LIN {X 0,Y 497.029,Z 1160.432,A -85,B 0,C 180,E1 21832.452,E2 21832.452} C_VEL
LIN {X 0,Y 502.234,Z 1141.982,A -85,B 0,C 180,E1 21830.218,E2 21830.218} C_VEL
LIN {X 0,Y 508.212,Z 1120.317,A -85,B 0,C 180,E1 21827.949,E2 21827.949} C_VEL
LIN {X 0,Y 512.986,Z 1102.562,A -85,B 0,C 180,E1 21826.314,E2 21826.314} C_VEL
LIN {X 0,Y 517.599,Z 1084.829,A -85,B 0,C 180,E1 21824.86,E2 21824.86} C_VEL
LIN {X 0,Y 522.261,Z 1066.052,A -85,B 0,C 180,E1 21823.491,E2 21823.491} C_VEL
LIN {X 0,Y 527.633,Z 1043.21,A -85,B 0,C 180,E1 21822.036,E2 21822.036} C_VEL
LIN {X 0,Y 533.047,Z 1017.477,A -85,B 0,C 180,E1 21820.656,E2 21820.656} C_VEL
LIN {X 0,Y 537.035,Z 996.541,A -85,B 0,C 180,E1 21819.707,E2 21819.707} C_VEL
LIN {X 0,Y 540.556,Z 975.901,A -85,B 0,C 180,E1 21818.909,E2 21818.909} C_VEL
LIN {X 0,Y 543.808,Z 954.173,A -85,B 0,C 180,E1 21818.206,E2 21818.206} C_VEL
LIN {X 0,Y 547.16,Z 927.563,A -85,B 0,C 180,E1 21817.516,E2 21817.516} C_VEL
LIN {X 0,Y 549.546,Z 900.175,A -85,B 0,C 180,E1 21816.999,E2 21816.999} C_VEL
LIN {X 0,Y 555.879,Z 766.866,A -85,B 0,C 180,E1 21814.975,E2 21814.975} C_VEL
LIN {X 0,Y 566.177,Z 554.638,A -85,B 0,C 180,E1 21811.749,E2 21811.749} C_VEL
LIN {X 0,Y 566.782,Z 540.369,A -85,B 0,C 180,E1 21811.512,E2 21811.512} C_VEL
LIN {X 0,Y 555.133,Z 521.953,A -85,B 0,C 180,E1 21809.04,E2 21809.04} C_VEL
LIN {X 0,Y 545.079,Z 507.132,A -85,B 0,C 180,E1 21806.678,E2 21806.678} C_VEL
LIN {X 0,Y 535.268,Z 493.183,A -85,B 0,C 180,E1 21804.09,E2 21804.09} C_VEL
LIN {X 0,Y 527.729,Z 483.129,A -85,B 0,C 180,E1 21801.858,E2 21801.858} C_VEL
LIN {X 0,Y 523.599,Z 477.699,A -85,B 0,C 180,E1 21800.513,E2 21800.513} C_VEL
LIN {X 0,Y 518.429,Z 471.033,A -85,B 0,C 180,E1 21798.673,E2 21798.673} C_VEL
LIN {X 0,Y 515.934,Z 468.011,A -85,B 0,C 180,E1 21797.714,E2 21797.714} C_VEL
LIN {X 0,Y 512.62,Z 464.186,A -85,B 0,C 180,E1 21796.352,E2 21796.352} C_VEL
LIN {X 0,Y 511.594,Z 462.527,A -85,B 0,C 180,E1 21795.88,E2 21795.88} C_VEL
LIN {X 0,Y 508.237,Z 459.547,A -85,B 0,C 180,E1 21794.353,E2 21794.353} C_VEL
LIN {X 0,Y 505.989,Z 456.089,A -85,B 0,C 180,E1 21793.135,E2 21793.135} C_VEL
LIN {X 0,Y 502.714,Z 453.695,A -85,B 0,C 180,E1 21791.298,E2 21791.298} C_VEL
LIN {X 0,Y 500.503,Z 449.64,A -85,B 0,C 180,E1 21789.661,E2 21789.661} C_VEL
LIN {X 0,Y 496.627,Z 447.233,A -85,B 0,C 180,E1 21786.358,E2 21786.358} C_VEL
LIN {X 0,Y 494.773,Z 443.193,A -85,B 0,C 180,E1 21783.302,E2 21783.302} C_VEL
LIN {X 0,Y 493.904,Z 442.834,A -85,B 0,C 180,E1 21780.464,E2 21780.464} C_VEL
LIN {X 0,Y 494.784,Z 443.176,A -85,B 0,C 180,E1 21776.176,E2 21776.176} C_VEL
LIN {X 0,Y 496.308,Z 446.772,A -85,B 0,C 180,E1 21773.522,E2 21773.522} C_VEL
LIN {X 0,Y 499.957,Z 449.46,A -85,B 0,C 180,E1 21770.212,E2 21770.212} C_VEL
LIN {X 0,Y 500.671,Z 449.883,A -85,B 0,C 180,E1 21769.704,E2 21769.704} C_VEL
LIN {X 0,Y 502.481,Z 453.39,A -85,B 0,C 180,E1 21768.347,E2 21768.347} C_VEL
LIN {X 0,Y 506.131,Z 456.157,A -85,B 0,C 180,E1 21766.286,E2 21766.286} C_VEL
LIN {X 0,Y 509.284,Z 460.773,A -85,B 0,C 180,E1 21764.63,E2 21764.63} C_VEL
LIN {X 0,Y 511.991,Z 463.084,A -85,B 0,C 180,E1 21763.433,E2 21763.433} C_VEL
LIN {X 0,Y 515.015,Z 467.149,A -85,B 0,C 180,E1 21762.136,E2 21762.136} C_VEL
LIN {X 0,Y 517.324,Z 469.281,A -85,B 0,C 180,E1 21761.256,E2 21761.256} C_VEL
LIN {X 0,Y 520.829,Z 473.673,A -85,B 0,C 180,E1 21759.959,E2 21759.959} C_VEL
LIN {X 0,Y 522.505,Z 475.511,A -85,B 0,C 180,E1 21759.383,E2 21759.383} C_VEL
LIN {X 0,Y 526.451,Z 480.194,A -85,B 0,C 180,E1 21758.086,E2 21758.086} C_VEL
LIN {X 0,Y 532.504,Z 487.779,A -85,B 0,C 180,E1 21756.248,E2 21756.248} C_VEL
LIN {X 0,Y 537.349,Z 493.885,A -85,B 0,C 180,E1 21754.896,E2 21754.896} C_VEL
LIN {X 0,Y 544.214,Z 502.496,A -85,B 0,C 180,E1 21753.129,E2 21753.129} C_VEL
LIN {X 0,Y 555.457,Z 517.635,A -85,B 0,C 180,E1 21750.506,E2 21750.506} C_VEL
LIN {X 0,Y 566.795,Z 533.76,A -85,B 0,C 180,E1 21748.135,E2 21748.135} C_VEL
LIN {X 0,Y 556.148,Z 750.221,A -85,B 0,C 180,E1 21744.845,E2 21744.845} C_VEL
LIN {X 0,Y 549.972,Z 878.471,A -85,B 0,C 180,E1 21742.897,E2 21742.897} C_VEL
LIN {X 0,Y 547.763,Z 904.531,A -85,B 0,C 180,E1 21742.395,E2 21742.395} C_VEL
LIN {X 0,Y 544.492,Z 931.574,A -85,B 0,C 180,E1 21741.681,E2 21741.681} C_VEL
LIN {X 0,Y 541.398,Z 952.771,A -85,B 0,C 180,E1 21740.982,E2 21740.982} C_VEL
LIN {X 0,Y 538.057,Z 972.694,A -85,B 0,C 180,E1 21740.201,E2 21740.201} C_VEL
LIN {X 0,Y 534.237,Z 992.896,A -85,B 0,C 180,E1 21739.277,E2 21739.277} C_VEL
LIN {X 0,Y 529.413,Z 1016.049,A -85,B 0,C 180,E1 21738.041,E2 21738.041} C_VEL
LIN {X 0,Y 523.704,Z 1040.347,A -85,B 0,C 180,E1 21736.501,E2 21736.501} C_VEL
LIN {X 0,Y 518.815,Z 1059.671,A -85,B 0,C 180,E1 21735.083,E2 21735.083} C_VEL
LIN {X 0,Y 514.02,Z 1077.682,A -85,B 0,C 180,E1 21733.587,E2 21733.587} C_VEL
LIN {X 0,Y 509.135,Z 1095.319,A -85,B 0,C 180,E1 21731.935,E2 21731.935} C_VEL
LIN {X 0,Y 503.229,Z 1115.953,A -85,B 0,C 180,E1 21729.74,E2 21729.74} C_VEL
LIN {X 0,Y 498.603,Z 1131.683,A -85,B 0,C 180,E1 21727.817,E2 21727.817} C_VEL
LIN {X 0,Y 496.227,Z 1136.911,A -85,B 0,C 180,E1 21727.204,E2 21727.204} C_VEL
LIN {X 0,Y 486.897,Z 1150.907,A -85,B 0,C 180,E1 21725.694,E2 21725.694} C_VEL
LIN {X 0,Y 485.066,Z 1155.035,A -85,B 0,C 180,E1 21725.127,E2 21725.127} C_VEL
LIN {X 0,Y 480.071,Z 1171.483,A -85,B 0,C 180,E1 21722.354,E2 21722.354} C_VEL
LIN {X 0,Y 476.443,Z 1184.012,A -85,B 0,C 180,E1 21719.957,E2 21719.957} C_VEL
LIN {X 0,Y 473.338,Z 1195.518,A -85,B 0,C 180,E1 21717.474,E2 21717.474} C_VEL
LIN {X 0,Y 470.207,Z 1208.206,A -85,B 0,C 180,E1 21714.357,E2 21714.357} C_VEL
LIN {X 0,Y 467.788,Z 1219.059,A -85,B 0,C 180,E1 21711.169,E2 21711.169} C_VEL
LIN {X 0,Y 466.306,Z 1226.894,A -85,B 0,C 180,E1 21708.496,E2 21708.496} C_VEL
LIN {X 0,Y 465.289,Z 1233.576,A -85,B 0,C 180,E1 21705.831,E2 21705.831} C_VEL
LIN {X 0,Y 464.545,Z 1239.653,A -85,B 0,C 180,E1 21702.929,E2 21702.929} C_VEL
LIN {X 0,Y 464.073,Z 1245.171,A -85,B 0,C 180,E1 21699.543,E2 21699.543} C_VEL
LIN {X 0,Y 463.961,Z 1248.712,A -85,B 0,C 180,E1 21696.529,E2 21696.529} C_VEL
LIN {X 0,Y 463.915,Z 1250.719,A -85,B 0,C 180,E1 21693.949,E2 21693.949} C_VEL
LIN {X 0,Y 463.904,Z 1251.727,A -85,B 0,C 180,E1 21691.476,E2 21691.476} C_VEL
LIN {X 0,Y 463.872,Z 1251.832,A -85,B 0,C 180,E1 21689.006,E2 21689.006} C_VEL
LIN {X 0,Y 463.913,Z 1251.035,A -85,B 0,C 180,E1 21686.535,E2 21686.535} C_VEL
LIN {X 0,Y 463.95,Z 1249.219,A -85,B 0,C 180,E1 21683.933,E2 21683.933} C_VEL
LIN {X 0,Y 464.051,Z 1246.391,A -85,B 0,C 180,E1 21681.32,E2 21681.32} C_VEL
LIN {X 0,Y 464.326,Z 1242,A -85,B 0,C 180,E1 21678.316,E2 21678.316} C_VEL
LIN {X 0,Y 465.026,Z 1235.477,A -85,B 0,C 180,E1 21674.892,E2 21674.892} C_VEL
LIN {X 0,Y 466.1,Z 1228.126,A -85,B 0,C 180,E1 21671.868,E2 21671.868} C_VEL
LIN {X 0,Y 467.52,Z 1220.38,A -85,B 0,C 180,E1 21669.167,E2 21669.167} C_VEL
LIN {X 0,Y 469.256,Z 1212.057,A -85,B 0,C 180,E1 21666.647,E2 21666.647} C_VEL
LIN {X 0,Y 471.63,Z 1202.142,A -85,B 0,C 180,E1 21664.016,E2 21664.016} C_VEL
LIN {X 0,Y 475.367,Z 1188.092,A -85,B 0,C 180,E1 21660.787,E2 21660.787} C_VEL
LIN {X 0,Y 479.151,Z 1174.611,A -85,B 0,C 180,E1 21658.128,E2 21658.128} C_VEL
LIN {X 0,Y 482.964,Z 1161.693,A -85,B 0,C 180,E1 21655.867,E2 21655.867} C_VEL
LIN {X 0,Y 487.08,Z 1148.162,A -85,B 0,C 180,E1 21653.753,E2 21653.753} C_VEL
LIN {X 0,Y 492.267,Z 1131.357,A -85,B 0,C 180,E1 21651.418,E2 21651.418} C_VEL
LIN {X 0,Y 498.504,Z 1110.82,A -85,B 0,C 180,E1 21648.954,E2 21648.954} C_VEL
LIN {X 0,Y 503.601,Z 1093.635,A -85,B 0,C 180,E1 21647.15,E2 21647.15} C_VEL
LIN {X 0,Y 508.295,Z 1077.31,A -85,B 0,C 180,E1 21645.624,E2 21645.624} C_VEL
LIN {X 0,Y 513.079,Z 1059.953,A -85,B 0,C 180,E1 21644.176,E2 21644.176} C_VEL
LIN {X 0,Y 518.353,Z 1039.81,A -85,B 0,C 180,E1 21642.694,E2 21642.694} C_VEL
LIN {X 0,Y 524.566,Z 1013.892,A -85,B 0,C 180,E1 21641.069,E2 21641.069} C_VEL
LIN {X 0,Y 529.021,Z 993.124,A -85,B 0,C 180,E1 21639.962,E2 21639.962} C_VEL
LIN {X 0,Y 532.958,Z 972.91,A -85,B 0,C 180,E1 21639.036,E2 21639.036} C_VEL
LIN {X 0,Y 536.564,Z 952.039,A -85,B 0,C 180,E1 21638.22,E2 21638.22} C_VEL
LIN {X 0,Y 540.132,Z 928.072,A -85,B 0,C 180,E1 21637.442,E2 21637.442} C_VEL
LIN {X 0,Y 543.36,Z 900.216,A -85,B 0,C 180,E1 21636.745,E2 21636.745} C_VEL
LIN {X 0,Y 545.306,Z 877.407,A -85,B 0,C 180,E1 21636.317,E2 21636.317} C_VEL
LIN {X 0,Y 555.554,Z 671.599,A -85,B 0,C 180,E1 21633.181,E2 21633.181} C_VEL
LIN {X 0,Y 562.367,Z 538.21,A -85,B 0,C 180,E1 21631.128,E2 21631.128} C_VEL
LIN {X 0,Y 551.699,Z 522.97,A -85,B 0,C 180,E1 21628.822,E2 21628.822} C_VEL
LIN {X 0,Y 541.383,Z 508.945,A -85,B 0,C 180,E1 21626.342,E2 21626.342} C_VEL
LIN {X 0,Y 532.518,Z 497.635,A -85,B 0,C 180,E1 21623.957,E2 21623.957} C_VEL
LIN {X 0,Y 528.303,Z 492.352,A -85,B 0,C 180,E1 21622.712,E2 21622.712} C_VEL
LIN {X 0,Y 524.222,Z 487.316,A -85,B 0,C 180,E1 21621.424,E2 21621.424} C_VEL
LIN {X 0,Y 519.631,Z 481.696,A -85,B 0,C 180,E1 21619.854,E2 21619.854} C_VEL
LIN {X 0,Y 515.928,Z 477.216,A -85,B 0,C 180,E1 21618.474,E2 21618.474} C_VEL
LIN {X 0,Y 514.556,Z 475.732,A -85,B 0,C 180,E1 21617.939,E2 21617.939} C_VEL
LIN {X 0,Y 511.083,Z 471.685,A -85,B 0,C 180,E1 21616.48,E2 21616.48} C_VEL
LIN {X 0,Y 509.897,Z 470.059,A -85,B 0,C 180,E1 21615.934,E2 21615.934} C_VEL
LIN {X 0,Y 506.547,Z 466.804,A -85,B 0,C 180,E1 21614.343,E2 21614.343} C_VEL
LIN {X 0,Y 504.877,Z 463.969,A -85,B 0,C 180,E1 21613.398,E2 21613.398} C_VEL
LIN {X 0,Y 501.485,Z 461.38,A -85,B 0,C 180,E1 21611.443,E2 21611.443} C_VEL
LIN {X 0,Y 499.477,Z 457.698,A -85,B 0,C 180,E1 21609.914,E2 21609.914} C_VEL
LIN {X 0,Y 495.09,Z 454.362,A -85,B 0,C 180,E1 21605.796,E2 21605.796} C_VEL
LIN {X 0,Y 493.761,Z 450.858,A -85,B 0,C 180,E1 21603.018,E2 21603.018} C_VEL
LIN {X 0,Y 493.831,Z 450.948,A -85,B 0,C 180,E1 21597.215,E2 21597.215} C_VEL
LIN {X 0,Y 495.777,Z 455.253,A -85,B 0,C 180,E1 21593.748,E2 21593.748} C_VEL
LIN {X 0,Y 499.49,Z 457.7,A -85,B 0,C 180,E1 21590.494,E2 21590.494} C_VEL
LIN {X 0,Y 501.581,Z 461.525,A -85,B 0,C 180,E1 21588.909,E2 21588.909} C_VEL
LIN {X 0,Y 505.181,Z 464.453,A -85,B 0,C 180,E1 21586.843,E2 21586.843} C_VEL
LIN {X 0,Y 507.875,Z 468.4,A -85,B 0,C 180,E1 21585.404,E2 21585.404} C_VEL
LIN {X 0,Y 510.518,Z 470.754,A -85,B 0,C 180,E1 21584.202,E2 21584.202} C_VEL
LIN {X 0,Y 513.616,Z 474.922,A -85,B 0,C 180,E1 21582.846,E2 21582.846} C_VEL
LIN {X 0,Y 515.651,Z 477.08,A -85,B 0,C 180,E1 21582.042,E2 21582.042} C_VEL
LIN {X 0,Y 519.586,Z 482.261,A -85,B 0,C 180,E1 21580.554,E2 21580.554} C_VEL
LIN {X 0,Y 523.665,Z 487.63,A -85,B 0,C 180,E1 21579.139,E2 21579.139} C_VEL
LIN {X 0,Y 528.756,Z 494.46,A -85,B 0,C 180,E1 21577.514,E2 21577.514} C_VEL
LIN {X 0,Y 534.895,Z 503.025,A -85,B 0,C 180,E1 21575.716,E2 21575.716} C_VEL
LIN {X 0,Y 543.878,Z 515.818,A -85,B 0,C 180,E1 21573.347,E2 21573.347} C_VEL
LIN {X 0,Y 554.813,Z 532.468,A -85,B 0,C 180,E1 21570.764,E2 21570.764} C_VEL
LIN {X 0,Y 562.515,Z 545.109,A -85,B 0,C 180,E1 21569.096,E2 21569.096} C_VEL
LIN {X 0,Y 551.791,Z 757.323,A -85,B 0,C 180,E1 21565.855,E2 21565.855} C_VEL
LIN {X 0,Y 544.786,Z 899.692,A -85,B 0,C 180,E1 21563.684,E2 21563.684} C_VEL
LIN {X 0,Y 542.427,Z 926.225,A -85,B 0,C 180,E1 21563.184,E2 21563.184} C_VEL
LIN {X 0,Y 538.96,Z 953.287,A -85,B 0,C 180,E1 21562.491,E2 21562.491} C_VEL
LIN {X 0,Y 535.662,Z 974.729,A -85,B 0,C 180,E1 21561.803,E2 21561.803} C_VEL
LIN {X 0,Y 532.026,Z 995.532,A -85,B 0,C 180,E1 21561.002,E2 21561.002} C_VEL
LIN {X 0,Y 527.885,Z 1016.607,A -85,B 0,C 180,E1 21560.05,E2 21560.05} C_VEL
LIN {X 0,Y 522.429,Z 1041.913,A -85,B 0,C 180,E1 21558.699,E2 21558.699} C_VEL
LIN {X 0,Y 516.806,Z 1065.056,A -85,B 0,C 180,E1 21557.227,E2 21557.227} C_VEL
LIN {X 0,Y 512.008,Z 1083.719,A -85,B 0,C 180,E1 21555.867,E2 21555.867} C_VEL
LIN {X 0,Y 507.226,Z 1101.42,A -85,B 0,C 180,E1 21554.415,E2 21554.415} C_VEL
LIN {X 0,Y 502.213,Z 1119.333,A -85,B 0,C 180,E1 21552.763,E2 21552.763} C_VEL
LIN {X 0,Y 496.243,Z 1140.304,A -85,B 0,C 180,E1 21550.569,E2 21550.569} C_VEL
LIN {X 0,Y 490.533,Z 1159.602,A -85,B 0,C 180,E1 21548.221,E2 21548.221} C_VEL
LIN {X 0,Y 486.187,Z 1174.525,A -85,B 0,C 180,E1 21546.178,E2 21546.178} C_VEL
LIN {X 0,Y 482.185,Z 1188.461,A -85,B 0,C 180,E1 21544.052,E2 21544.052} C_VEL
LIN {X 0,Y 478.313,Z 1202.513,A -85,B 0,C 180,E1 21541.653,E2 21541.653} C_VEL
LIN {X 0,Y 473.954,Z 1219.168,A -85,B 0,C 180,E1 21538.389,E2 21538.389} C_VEL
LIN {X 0,Y 471.191,Z 1230.65,A -85,B 0,C 180,E1 21535.791,E2 21535.791} C_VEL
LIN {X 0,Y 468.998,Z 1240.65,A -85,B 0,C 180,E1 21533.234,E2 21533.234} C_VEL
LIN {X 0,Y 467.323,Z 1249.445,A -85,B 0,C 180,E1 21530.678,E2 21530.678} C_VEL
LIN {X 0,Y 465.884,Z 1258.181,A -85,B 0,C 180,E1 21527.749,E2 21527.749} C_VEL
LIN {X 0,Y 464.794,Z 1266.563,A -85,B 0,C 180,E1 21524.328,E2 21524.328} C_VEL
LIN {X 0,Y 464.305,Z 1272.056,A -85,B 0,C 180,E1 21521.52,E2 21521.52} C_VEL
LIN {X 0,Y 464.051,Z 1276.014,A -85,B 0,C 180,E1 21518.93,E2 21518.93} C_VEL
LIN {X 0,Y 463.958,Z 1278.95,A -85,B 0,C 180,E1 21516.316,E2 21516.316} C_VEL
LIN {X 0,Y 463.916,Z 1280.806,A -85,B 0,C 180,E1 21513.836,E2 21513.836} C_VEL
LIN {X 0,Y 463.896,Z 1281.756,A -85,B 0,C 180,E1 21511.364,E2 21511.364} C_VEL
LIN {X 0,Y 463.881,Z 1281.803,A -85,B 0,C 180,E1 21508.894,E2 21508.894} C_VEL
LIN {X 0,Y 463.913,Z 1280.948,A -85,B 0,C 180,E1 21506.422,E2 21506.422} C_VEL
LIN {X 0,Y 463.949,Z 1279.187,A -85,B 0,C 180,E1 21503.944,E2 21503.944} C_VEL
LIN {X 0,Y 464.051,Z 1276.347,A -85,B 0,C 180,E1 21501.331,E2 21501.331} C_VEL
LIN {X 0,Y 464.262,Z 1272.648,A -85,B 0,C 180,E1 21498.83,E2 21498.83} C_VEL
LIN {X 0,Y 464.68,Z 1267.896,A -85,B 0,C 180,E1 21496.315,E2 21496.315} C_VEL
LIN {X 0,Y 465.38,Z 1261.818,A -85,B 0,C 180,E1 21493.66,E2 21493.66} C_VEL
LIN {X 0,Y 466.562,Z 1253.866,A -85,B 0,C 180,E1 21490.736,E2 21490.736} C_VEL
LIN {X 0,Y 468.621,Z 1242.575,A -85,B 0,C 180,E1 21487.289,E2 21487.289} C_VEL
LIN {X 0,Y 470.829,Z 1232.284,A -85,B 0,C 180,E1 21484.605,E2 21484.605} C_VEL
LIN {X 0,Y 473.308,Z 1221.766,A -85,B 0,C 180,E1 21482.176,E2 21482.176} C_VEL
LIN {X 0,Y 476.286,Z 1209.997,A -85,B 0,C 180,E1 21479.754,E2 21479.754} C_VEL
LIN {X 0,Y 480.497,Z 1194.732,A -85,B 0,C 180,E1 21476.97,E2 21476.97} C_VEL
LIN {X 0,Y 485.421,Z 1177.178,A -85,B 0,C 180,E1 21474.206,E2 21474.206} C_VEL
LIN {X 0,Y 489.946,Z 1161.563,A -85,B 0,C 180,E1 21472.035,E2 21472.035} C_VEL
LIN {X 0,Y 494.553,Z 1145.778,A -85,B 0,C 180,E1 21470.074,E2 21470.074} C_VEL
LIN {X 0,Y 500.556,Z 1125.32,A -85,B 0,C 180,E1 21467.825,E2 21467.825} C_VEL
LIN {X 0,Y 506.453,Z 1104.21,A -85,B 0,C 180,E1 21465.829,E2 21465.829} C_VEL
LIN {X 0,Y 511.371,Z 1086.037,A -85,B 0,C 180,E1 21464.315,E2 21464.315} C_VEL
LIN {X 0,Y 516.177,Z 1067.413,A -85,B 0,C 180,E1 21462.938,E2 21462.938} C_VEL
LIN {X 0,Y 521.032,Z 1047.472,A -85,B 0,C 180,E1 21461.64,E2 21461.64} C_VEL
LIN {X 0,Y 526.618,Z 1022.881,A -85,B 0,C 180,E1 21460.258,E2 21460.258} C_VEL
LIN {X 0,Y 531.493,Z 998.254,A -85,B 0,C 180,E1 21459.114,E2 21459.114} C_VEL
LIN {X 0,Y 535.242,Z 977.114,A -85,B 0,C 180,E1 21458.285,E2 21458.285} C_VEL
LIN {X 0,Y 538.532,Z 955.967,A -85,B 0,C 180,E1 21457.591,E2 21457.591} C_VEL
LIN {X 0,Y 541.423,Z 934.088,A -85,B 0,C 180,E1 21457.003,E2 21457.003} C_VEL
LIN {X 0,Y 544.311,Z 906.44,A -85,B 0,C 180,E1 21456.43,E2 21456.43} C_VEL
LIN {X 0,Y 546.777,Z 860.87,A -85,B 0,C 180,E1 21455.715,E2 21455.715} C_VEL
LIN {X 0,Y 557.422,Z 642.939,A -85,B 0,C 180,E1 21452.406,E2 21452.406} C_VEL
LIN {X 0,Y 562.394,Z 544.765,A -85,B 0,C 180,E1 21450.889,E2 21450.889} C_VEL
LIN {X 0,Y 551.819,Z 527.929,A -85,B 0,C 180,E1 21448.579,E2 21448.579} C_VEL
LIN {X 0,Y 542.426,Z 513.869,A -85,B 0,C 180,E1 21446.317,E2 21446.317} C_VEL
LIN {X 0,Y 532.943,Z 500.218,A -85,B 0,C 180,E1 21443.76,E2 21443.76} C_VEL
LIN {X 0,Y 525.603,Z 490.294,A -85,B 0,C 180,E1 21441.54,E2 21441.54} C_VEL
LIN {X 0,Y 521.54,Z 484.891,A -85,B 0,C 180,E1 21440.188,E2 21440.188} C_VEL
LIN {X 0,Y 516.605,Z 478.402,A -85,B 0,C 180,E1 21438.39,E2 21438.39} C_VEL
LIN {X 0,Y 514.143,Z 475.469,A -85,B 0,C 180,E1 21437.427,E2 21437.427} C_VEL
LIN {X 0,Y 510.824,Z 471.415,A -85,B 0,C 180,E1 21436.021,E2 21436.021} C_VEL
LIN {X 0,Y 509.874,Z 470.095,A -85,B 0,C 180,E1 21435.585,E2 21435.585} C_VEL
LIN {X 0,Y 506.394,Z 466.67,A -85,B 0,C 180,E1 21433.939,E2 21433.939} C_VEL
LIN {X 0,Y 504.598,Z 463.872,A -85,B 0,C 180,E1 21432.939,E2 21432.939} C_VEL
LIN {X 0,Y 501.39,Z 461.389,A -85,B 0,C 180,E1 21431.095,E2 21431.095} C_VEL
LIN {X 0,Y 499.213,Z 457.481,A -85,B 0,C 180,E1 21429.453,E2 21429.453} C_VEL
LIN {X 0,Y 495.356,Z 454.892,A -85,B 0,C 180,E1 21426.025,E2 21426.025} C_VEL
LIN {X 0,Y 493.629,Z 450.851,A -85,B 0,C 180,E1 21422.903,E2 21422.903} C_VEL
LIN {X 0,Y 493.719,Z 450.879,A -85,B 0,C 180,E1 21416.4,E2 21416.4} C_VEL
LIN {X 0,Y 495.239,Z 454.651,A -85,B 0,C 180,E1 21413.624,E2 21413.624} C_VEL
LIN {X 0,Y 498.995,Z 457.415,A -85,B 0,C 180,E1 21410.193,E2 21410.193} C_VEL
LIN {X 0,Y 499.518,Z 457.987,A -85,B 0,C 180,E1 21409.796,E2 21409.796} C_VEL
LIN {X 0,Y 501.418,Z 461.402,A -85,B 0,C 180,E1 21408.381,E2 21408.381} C_VEL
LIN {X 0,Y 505.141,Z 464.462,A -85,B 0,C 180,E1 21406.259,E2 21406.259} C_VEL
LIN {X 0,Y 507.741,Z 468.347,A -85,B 0,C 180,E1 21404.875,E2 21404.875} C_VEL
LIN {X 0,Y 510.458,Z 470.765,A -85,B 0,C 180,E1 21403.645,E2 21403.645} C_VEL
LIN {X 0,Y 513.648,Z 474.968,A -85,B 0,C 180,E1 21402.263,E2 21402.263} C_VEL
LIN {X 0,Y 515.651,Z 476.867,A -85,B 0,C 180,E1 21401.487,E2 21401.487} C_VEL
LIN {X 0,Y 519.419,Z 481.504,A -85,B 0,C 180,E1 21400.079,E2 21400.079} C_VEL
LIN {X 0,Y 521.209,Z 483.769,A -85,B 0,C 180,E1 21399.447,E2 21399.447} C_VEL
LIN {X 0,Y 525.787,Z 489.279,A -85,B 0,C 180,E1 21397.939,E2 21397.939} C_VEL
LIN {X 0,Y 530.484,Z 495.159,A -85,B 0,C 180,E1 21396.506,E2 21396.506} C_VEL
LIN {X 0,Y 535.454,Z 501.51,A -85,B 0,C 180,E1 21395.096,E2 21395.096} C_VEL
LIN {X 0,Y 541.963,Z 509.803,A -85,B 0,C 180,E1 21393.393,E2 21393.393} C_VEL
LIN {X 0,Y 552.775,Z 524.522,A -85,B 0,C 180,E1 21390.824,E2 21390.824} C_VEL
LIN {X 0,Y 562.381,Z 538.342,A -85,B 0,C 180,E1 21388.762,E2 21388.762} C_VEL
LIN {X 0,Y 551.332,Z 755.458,A -85,B 0,C 180,E1 21385.45,E2 21385.45} C_VEL
LIN {X 0,Y 545.179,Z 878.788,A -85,B 0,C 180,E1 21383.567,E2 21383.567} C_VEL
LIN {X 0,Y 542.874,Z 905.198,A -85,B 0,C 180,E1 21383.056,E2 21383.056} C_VEL
LIN {X 0,Y 539.515,Z 932.066,A -85,B 0,C 180,E1 21382.344,E2 21382.344} C_VEL
LIN {X 0,Y 536.337,Z 953.216,A -85,B 0,C 180,E1 21381.644,E2 21381.644} C_VEL
LIN {X 0,Y 532.92,Z 972.969,A -85,B 0,C 180,E1 21380.868,E2 21380.868} C_VEL
LIN {X 0,Y 528.987,Z 993.17,A -85,B 0,C 180,E1 21379.942,E2 21379.942} C_VEL
LIN {X 0,Y 524.098,Z 1015.92,A -85,B 0,C 180,E1 21378.725,E2 21378.725} C_VEL
LIN {X 0,Y 518.113,Z 1040.621,A -85,B 0,C 180,E1 21377.157,E2 21377.157} C_VEL
LIN {X 0,Y 513.081,Z 1059.873,A -85,B 0,C 180,E1 21375.737,E2 21375.737} C_VEL
LIN {X 0,Y 508.2,Z 1077.578,A -85,B 0,C 180,E1 21374.26,E2 21374.26} C_VEL
LIN {X 0,Y 503.244,Z 1094.82,A -85,B 0,C 180,E1 21372.641,E2 21372.641} C_VEL
LIN {X 0,Y 497.273,Z 1115.029,A -85,B 0,C 180,E1 21370.492,E2 21370.492} C_VEL
LIN {X 0,Y 491.355,Z 1134.185,A -85,B 0,C 180,E1 21368.114,E2 21368.114} C_VEL
LIN {X 0,Y 486.957,Z 1148.549,A -85,B 0,C 180,E1 21366.099,E2 21366.099} C_VEL
LIN {X 0,Y 485.066,Z 1155.035,A -85,B 0,C 180,E1 21365.127,E2 21365.127} C_VEL
LIN {X 0,Y 482.811,Z 1159.814,A -85,B 0,C 180,E1 21364.453,E2 21364.453} C_VEL
LIN {X 0,Y 473.489,Z 1172.374,A -85,B 0,C 180,E1 21362.728,E2 21362.728} C_VEL
LIN {X 0,Y 471.727,Z 1176.083,A -85,B 0,C 180,E1 21362.093,E2 21362.093} C_VEL
LIN {X 0,Y 466.996,Z 1192.12,A -85,B 0,C 180,E1 21358.791,E2 21358.791} C_VEL
LIN {X 0,Y 463.883,Z 1203.454,A -85,B 0,C 180,E1 21356.078,E2 21356.078} C_VEL
LIN {X 0,Y 461.498,Z 1212.969,A -85,B 0,C 180,E1 21353.487,E2 21353.487} C_VEL
LIN {X 0,Y 459.581,Z 1221.703,A -85,B 0,C 180,E1 21350.764,E2 21350.764} C_VEL
LIN {X 0,Y 457.834,Z 1231.194,A -85,B 0,C 180,E1 21347.272,E2 21347.272} C_VEL
LIN {X 0,Y 456.817,Z 1238.006,A -85,B 0,C 180,E1 21344.152,E2 21344.152} C_VEL
LIN {X 0,Y 456.332,Z 1242.744,A -85,B 0,C 180,E1 21341.495,E2 21341.495} C_VEL
LIN {X 0,Y 456.063,Z 1246.512,A -85,B 0,C 180,E1 21338.822,E2 21338.822} C_VEL
LIN {X 0,Y 455.957,Z 1249.28,A -85,B 0,C 180,E1 21336.162,E2 21336.162} C_VEL
LIN {X 0,Y 455.914,Z 1251.069,A -85,B 0,C 180,E1 21333.515,E2 21333.515} C_VEL
LIN {X 0,Y 455.872,Z 1251.893,A -85,B 0,C 180,E1 21330.874,E2 21330.874} C_VEL
LIN {X 0,Y 455.91,Z 1251.73,A -85,B 0,C 180,E1 21328.109,E2 21328.109} C_VEL
LIN {X 0,Y 455.928,Z 1250.234,A -85,B 0,C 180,E1 21324.836,E2 21324.836} C_VEL
LIN {X 0,Y 456.037,Z 1247.074,A -85,B 0,C 180,E1 21321.547,E2 21321.547} C_VEL
LIN {X 0,Y 456.285,Z 1243.268,A -85,B 0,C 180,E1 21318.748,E2 21318.748} C_VEL
LIN {X 0,Y 456.739,Z 1238.835,A -85,B 0,C 180,E1 21316.19,E2 21316.19} C_VEL
LIN {X 0,Y 457.498,Z 1233.141,A -85,B 0,C 180,E1 21313.489,E2 21313.489} C_VEL
LIN {X 0,Y 458.69,Z 1226.182,A -85,B 0,C 180,E1 21310.716,E2 21310.716} C_VEL
LIN {X 0,Y 460.854,Z 1215.914,A -85,B 0,C 180,E1 21307.277,E2 21307.277} C_VEL
LIN {X 0,Y 463.428,Z 1205.242,A -85,B 0,C 180,E1 21304.294,E2 21304.294} C_VEL
LIN {X 0,Y 466.258,Z 1194.672,A -85,B 0,C 180,E1 21301.705,E2 21301.705} C_VEL
LIN {X 0,Y 469.504,Z 1183.381,A -85,B 0,C 180,E1 21299.257,E2 21299.257} C_VEL
LIN {X 0,Y 473.822,Z 1169.379,A -85,B 0,C 180,E1 21296.575,E2 21296.575} C_VEL
LIN {X 0,Y 479.329,Z 1151.758,A -85,B 0,C 180,E1 21293.666,E2 21293.666} C_VEL
LIN {X 0,Y 484.037,Z 1136.973,A -85,B 0,C 180,E1 21291.528,E2 21291.528} C_VEL
LIN {X 0,Y 488.992,Z 1121.398,A -85,B 0,C 180,E1 21289.523,E2 21289.523} C_VEL
LIN {X 0,Y 494.706,Z 1103.27,A -85,B 0,C 180,E1 21287.458,E2 21287.458} C_VEL
LIN {X 0,Y 501.481,Z 1080.877,A -85,B 0,C 180,E1 21285.26,E2 21285.26} C_VEL
LIN {X 0,Y 506.836,Z 1062.205,A -85,B 0,C 180,E1 21283.669,E2 21283.669} C_VEL
LIN {X 0,Y 511.758,Z 1044.093,A -85,B 0,C 180,E1 21282.305,E2 21282.305} C_VEL
LIN {X 0,Y 516.855,Z 1024.083,A -85,B 0,C 180,E1 21280.982,E2 21280.982} C_VEL
LIN {X 0,Y 522.699,Z 998.992,A -85,B 0,C 180,E1 21279.56,E2 21279.56} C_VEL
LIN {X 0,Y 527.427,Z 975.719,A -85,B 0,C 180,E1 21278.464,E2 21278.464} C_VEL
LIN {X 0,Y 531.208,Z 954.707,A -85,B 0,C 180,E1 21277.626,E2 21277.626} C_VEL
LIN {X 0,Y 534.427,Z 934.083,A -85,B 0,C 180,E1 21276.934,E2 21276.934} C_VEL
LIN {X 0,Y 537.436,Z 911.189,A -85,B 0,C 180,E1 21276.307,E2 21276.307} C_VEL
LIN {X 0,Y 540.316,Z 881.853,A -85,B 0,C 180,E1 21275.702,E2 21275.702} C_VEL
LIN {X 0,Y 543.364,Z 825.579,A -85,B 0,C 180,E1 21274.827,E2 21274.827} C_VEL
LIN {X 0,Y 554.655,Z 606.621,A -85,B 0,C 180,E1 21271.485,E2 21271.485} C_VEL
LIN {X 0,Y 558.058,Z 542.861,A -85,B 0,C 180,E1 21270.498,E2 21270.498} C_VEL
LIN {X 0,Y 548.432,Z 529.017,A -85,B 0,C 180,E1 21268.355,E2 21268.355} C_VEL
LIN {X 0,Y 538.87,Z 515.862,A -85,B 0,C 180,E1 21266,E2 21266} C_VEL
LIN {X 0,Y 530.138,Z 504.583,A -85,B 0,C 180,E1 21263.599,E2 21263.599} C_VEL
LIN {X 0,Y 526.158,Z 499.53,A -85,B 0,C 180,E1 21262.397,E2 21262.397} C_VEL
LIN {X 0,Y 522.298,Z 494.702,A -85,B 0,C 180,E1 21261.154,E2 21261.154} C_VEL
LIN {X 0,Y 517.772,Z 489.11,A -85,B 0,C 180,E1 21259.576,E2 21259.576} C_VEL
LIN {X 0,Y 514.007,Z 484.367,A -85,B 0,C 180,E1 21258.134,E2 21258.134} C_VEL
LIN {X 0,Y 509.732,Z 479.607,A -85,B 0,C 180,E1 21256.349,E2 21256.349} C_VEL
LIN {X 0,Y 508.446,Z 477.777,A -85,B 0,C 180,E1 21255.747,E2 21255.747} C_VEL
LIN {X 0,Y 505.043,Z 474.35,A -85,B 0,C 180,E1 21254.094,E2 21254.094} C_VEL
LIN {X 0,Y 503.495,Z 471.748,A -85,B 0,C 180,E1 21253.202,E2 21253.202} C_VEL
LIN {X 0,Y 500.09,Z 468.973,A -85,B 0,C 180,E1 21251.183,E2 21251.183} C_VEL
LIN {X 0,Y 498.054,Z 465.345,A -85,B 0,C 180,E1 21249.592,E2 21249.592} C_VEL
LIN {X 0,Y 494.112,Z 462.368,A -85,B 0,C 180,E1 21245.807,E2 21245.807} C_VEL
LIN {X 0,Y 492.74,Z 458.792,A -85,B 0,C 180,E1 21242.908,E2 21242.908} C_VEL
LIN {X 0,Y 492.839,Z 459.035,A -85,B 0,C 180,E1 21237.209,E2 21237.209} C_VEL
LIN {X 0,Y 494.802,Z 463.24,A -85,B 0,C 180,E1 21233.735,E2 21233.735} C_VEL
LIN {X 0,Y 498.283,Z 465.591,A -85,B 0,C 180,E1 21230.646,E2 21230.646} C_VEL
LIN {X 0,Y 500.349,Z 469.324,A -85,B 0,C 180,E1 21229.056,E2 21229.056} C_VEL
LIN {X 0,Y 503.8,Z 472.201,A -85,B 0,C 180,E1 21227.038,E2 21227.038} C_VEL
LIN {X 0,Y 506.679,Z 476.321,A -85,B 0,C 180,E1 21225.485,E2 21225.485} C_VEL
LIN {X 0,Y 509.051,Z 478.526,A -85,B 0,C 180,E1 21224.389,E2 21224.389} C_VEL
LIN {X 0,Y 512.386,Z 482.862,A -85,B 0,C 180,E1 21222.921,E2 21222.921} C_VEL
LIN {X 0,Y 514.395,Z 485.169,A -85,B 0,C 180,E1 21222.114,E2 21222.114} C_VEL
LIN {X 0,Y 518.016,Z 490.037,A -85,B 0,C 180,E1 21220.727,E2 21220.727} C_VEL
LIN {X 0,Y 521.823,Z 495.112,A -85,B 0,C 180,E1 21219.385,E2 21219.385} C_VEL
LIN {X 0,Y 528.11,Z 503.573,A -85,B 0,C 180,E1 21217.367,E2 21217.367} C_VEL
LIN {X 0,Y 536.711,Z 516.005,A -85,B 0,C 180,E1 21214.894,E2 21214.894} C_VEL
LIN {X 0,Y 544.517,Z 527.655,A -85,B 0,C 180,E1 21212.88,E2 21212.88} C_VEL
LIN {X 0,Y 553.47,Z 541.562,A -85,B 0,C 180,E1 21210.776,E2 21210.776} C_VEL
LIN {X 0,Y 558.165,Z 549.493,A -85,B 0,C 180,E1 21209.735,E2 21209.735} C_VEL
LIN {X 0,Y 547.088,Z 761.48,A -85,B 0,C 180,E1 21206.486,E2 21206.486} C_VEL
LIN {X 0,Y 540.058,Z 899.447,A -85,B 0,C 180,E1 21204.373,E2 21204.373} C_VEL
LIN {X 0,Y 537.611,Z 926.233,A -85,B 0,C 180,E1 21203.866,E2 21203.866} C_VEL
LIN {X 0,Y 534.058,Z 953.118,A -85,B 0,C 180,E1 21203.177,E2 21203.177} C_VEL
LIN {X 0,Y 530.677,Z 974.471,A -85,B 0,C 180,E1 21202.493,E2 21202.493} C_VEL
LIN {X 0,Y 526.933,Z 995.27,A -85,B 0,C 180,E1 21201.691,E2 21201.691} C_VEL
LIN {X 0,Y 522.8,Z 1015.667,A -85,B 0,C 180,E1 21200.772,E2 21200.772} C_VEL
LIN {X 0,Y 517.514,Z 1039.621,A -85,B 0,C 180,E1 21199.501,E2 21199.501} C_VEL
LIN {X 0,Y 511.494,Z 1063.771,A -85,B 0,C 180,E1 21197.978,E2 21197.978} C_VEL
LIN {X 0,Y 506.453,Z 1082.708,A -85,B 0,C 180,E1 21196.601,E2 21196.601} C_VEL
LIN {X 0,Y 501.484,Z 1100.455,A -85,B 0,C 180,E1 21195.145,E2 21195.145} C_VEL
LIN {X 0,Y 496.353,Z 1118.12,A -85,B 0,C 180,E1 21193.513,E2 21193.513} C_VEL
LIN {X 0,Y 490.596,Z 1137.526,A -85,B 0,C 180,E1 21191.486,E2 21191.486} C_VEL
LIN {X 0,Y 484.247,Z 1158.344,A -85,B 0,C 180,E1 21188.969,E2 21188.969} C_VEL
LIN {X 0,Y 479.395,Z 1174.25,A -85,B 0,C 180,E1 21186.774,E2 21186.774} C_VEL
LIN {X 0,Y 475.213,Z 1188.185,A -85,B 0,C 180,E1 21184.622,E2 21184.622} C_VEL
LIN {X 0,Y 471.002,Z 1202.701,A -85,B 0,C 180,E1 21182.109,E2 21182.109} C_VEL
LIN {X 0,Y 466.502,Z 1219.087,A -85,B 0,C 180,E1 21178.838,E2 21178.838} C_VEL
LIN {X 0,Y 463.5,Z 1230.9,A -85,B 0,C 180,E1 21176.114,E2 21176.114} C_VEL
LIN {X 0,Y 461.322,Z 1240.376,A -85,B 0,C 180,E1 21173.644,E2 21173.644} C_VEL
LIN {X 0,Y 459.533,Z 1249.251,A -85,B 0,C 180,E1 21171.019,E2 21171.019} C_VEL
LIN {X 0,Y 457.961,Z 1258.271,A -85,B 0,C 180,E1 21167.935,E2 21167.935} C_VEL
LIN {X 0,Y 456.852,Z 1266.294,A -85,B 0,C 180,E1 21164.583,E2 21164.583} C_VEL
LIN {X 0,Y 456.341,Z 1271.724,A -85,B 0,C 180,E1 21161.763,E2 21161.763} C_VEL
LIN {X 0,Y 456.051,Z 1275.807,A -85,B 0,C 180,E1 21159.088,E2 21159.088} C_VEL
LIN {X 0,Y 455.96,Z 1278.834,A -85,B 0,C 180,E1 21156.427,E2 21156.427} C_VEL
LIN {X 0,Y 455.917,Z 1280.749,A -85,B 0,C 180,E1 21153.904,E2 21153.904} C_VEL
LIN {X 0,Y 455.897,Z 1281.729,A -85,B 0,C 180,E1 21151.388,E2 21151.388} C_VEL
LIN {X 0,Y 455.875,Z 1281.8,A -85,B 0,C 180,E1 21149,E2 21149} C_VEL
LIN {X 0,Y 455.913,Z 1280.965,A -85,B 0,C 180,E1 21146.485,E2 21146.485} C_VEL
LIN {X 0,Y 455.948,Z 1279.195,A -85,B 0,C 180,E1 21143.964,E2 21143.964} C_VEL
LIN {X 0,Y 456.051,Z 1276.316,A -85,B 0,C 180,E1 21141.305,E2 21141.305} C_VEL
LIN {X 0,Y 456.284,Z 1272.381,A -85,B 0,C 180,E1 21138.632,E2 21138.632} C_VEL
LIN {X 0,Y 456.72,Z 1267.627,A -85,B 0,C 180,E1 21136.072,E2 21136.072} C_VEL
LIN {X 0,Y 457.477,Z 1261.548,A -85,B 0,C 180,E1 21133.369,E2 21133.369} C_VEL
LIN {X 0,Y 458.789,Z 1253.231,A -85,B 0,C 180,E1 21130.264,E2 21130.264} C_VEL
LIN {X 0,Y 460.916,Z 1242.3,A -85,B 0,C 180,E1 21126.888,E2 21126.888} C_VEL
LIN {X 0,Y 463.251,Z 1232.008,A -85,B 0,C 180,E1 21124.159,E2 21124.159} C_VEL
LIN {X 0,Y 465.941,Z 1221.181,A -85,B 0,C 180,E1 21121.624,E2 21121.624} C_VEL
LIN {X 0,Y 469.207,Z 1209.072,A -85,B 0,C 180,E1 21119.106,E2 21119.106} C_VEL
LIN {X 0,Y 473.844,Z 1192.957,A -85,B 0,C 180,E1 21116.155,E2 21116.155} C_VEL
LIN {X 0,Y 478.847,Z 1176.04,A -85,B 0,C 180,E1 21113.489,E2 21113.489} C_VEL
LIN {X 0,Y 483.468,Z 1160.814,A -85,B 0,C 180,E1 21111.358,E2 21111.358} C_VEL
LIN {X 0,Y 488.453,Z 1144.471,A -85,B 0,C 180,E1 21109.318,E2 21109.318} C_VEL
LIN {X 0,Y 494.842,Z 1123.428,A -85,B 0,C 180,E1 21107.01,E2 21107.01} C_VEL
LIN {X 0,Y 500.87,Z 1102.581,A -85,B 0,C 180,E1 21105.044,E2 21105.044} C_VEL
LIN {X 0,Y 505.764,Z 1085.145,A -85,B 0,C 180,E1 21103.592,E2 21103.592} C_VEL
LIN {X 0,Y 510.575,Z 1067.137,A -85,B 0,C 180,E1 21102.258,E2 21102.258} C_VEL
LIN {X 0,Y 515.363,Z 1048.104,A -85,B 0,C 180,E1 21101.01,E2 21101.01} C_VEL
LIN {X 0,Y 520.634,Z 1025.661,A -85,B 0,C 180,E1 21099.733,E2 21099.733} C_VEL
LIN {X 0,Y 526.14,Z 999.272,A -85,B 0,C 180,E1 21098.478,E2 21098.478} C_VEL
LIN {X 0,Y 530.116,Z 977.583,A -85,B 0,C 180,E1 21097.622,E2 21097.622} C_VEL
LIN {X 0,Y 533.599,Z 955.91,A -85,B 0,C 180,E1 21096.909,E2 21096.909} C_VEL
LIN {X 0,Y 536.544,Z 934.255,A -85,B 0,C 180,E1 21096.326,E2 21096.326} C_VEL
LIN {X 0,Y 539.517,Z 906.913,A -85,B 0,C 180,E1 21095.754,E2 21095.754} C_VEL
LIN {X 0,Y 542.043,Z 862.028,A -85,B 0,C 180,E1 21095.045,E2 21095.045} C_VEL
LIN {X 0,Y 553.058,Z 644.249,A -85,B 0,C 180,E1 21091.725,E2 21091.725} C_VEL
LIN {X 0,Y 558.072,Z 549.209,A -85,B 0,C 180,E1 21090.257,E2 21090.257} C_VEL
LIN {X 0,Y 548.247,Z 533.437,A -85,B 0,C 180,E1 21088.043,E2 21088.043} C_VEL
LIN {X 0,Y 539.323,Z 519.899,A -85,B 0,C 180,E1 21085.829,E2 21085.829} C_VEL
LIN {X 0,Y 530.373,Z 506.915,A -85,B 0,C 180,E1 21083.352,E2 21083.352} C_VEL
LIN {X 0,Y 523.494,Z 497.456,A -85,B 0,C 180,E1 21081.22,E2 21081.22} C_VEL
LIN {X 0,Y 519.498,Z 492.076,A -85,B 0,C 180,E1 21079.86,E2 21079.86} C_VEL
LIN {X 0,Y 514.794,Z 485.772,A -85,B 0,C 180,E1 21078.106,E2 21078.106} C_VEL
LIN {X 0,Y 512.501,Z 483.037,A -85,B 0,C 180,E1 21077.192,E2 21077.192} C_VEL
LIN {X 0,Y 509.122,Z 478.774,A -85,B 0,C 180,E1 21075.725,E2 21075.725} C_VEL
LIN {X 0,Y 508.17,Z 477.639,A -85,B 0,C 180,E1 21075.288,E2 21075.288} C_VEL
LIN {X 0,Y 504.683,Z 473.915,A -85,B 0,C 180,E1 21073.578,E2 21073.578} C_VEL
LIN {X 0,Y 503.214,Z 471.65,A -85,B 0,C 180,E1 21072.742,E2 21072.742} C_VEL
LIN {X 0,Y 499.99,Z 468.971,A -85,B 0,C 180,E1 21070.835,E2 21070.835} C_VEL
LIN {X 0,Y 497.93,Z 465.316,A -85,B 0,C 180,E1 21069.245,E2 21069.245} C_VEL
LIN {X 0,Y 494.193,Z 462.653,A -85,B 0,C 180,E1 21065.806,E2 21065.806} C_VEL
LIN {X 0,Y 492.602,Z 458.786,A -85,B 0,C 180,E1 21062.792,E2 21062.792} C_VEL
LIN {X 0,Y 492.728,Z 458.967,A -85,B 0,C 180,E1 21056.393,E2 21056.393} C_VEL
LIN {X 0,Y 494.171,Z 462.53,A -85,B 0,C 180,E1 21053.727,E2 21053.727} C_VEL
LIN {X 0,Y 497.874,Z 465.31,A -85,B 0,C 180,E1 21050.288,E2 21050.288} C_VEL
LIN {X 0,Y 498.372,Z 466.051,A -85,B 0,C 180,E1 21049.889,E2 21049.889} C_VEL
LIN {X 0,Y 500.445,Z 469.495,A -85,B 0,C 180,E1 21048.358,E2 21048.358} C_VEL
LIN {X 0,Y 503.753,Z 472.212,A -85,B 0,C 180,E1 21046.454,E2 21046.454} C_VEL
LIN {X 0,Y 506.545,Z 476.271,A -85,B 0,C 180,E1 21044.955,E2 21044.955} C_VEL
LIN {X 0,Y 508.938,Z 478.441,A -85,B 0,C 180,E1 21043.857,E2 21043.857} C_VEL
LIN {X 0,Y 512.285,Z 482.782,A -85,B 0,C 180,E1 21042.39,E2 21042.39} C_VEL
LIN {X 0,Y 514.12,Z 484.658,A -85,B 0,C 180,E1 21041.664,E2 21041.664} C_VEL
LIN {X 0,Y 518.012,Z 489.332,A -85,B 0,C 180,E1 21040.199,E2 21040.199} C_VEL
LIN {X 0,Y 523.997,Z 496.877,A -85,B 0,C 180,E1 21038.155,E2 21038.155} C_VEL
LIN {X 0,Y 528.644,Z 502.77,A -85,B 0,C 180,E1 21036.715,E2 21036.715} C_VEL
LIN {X 0,Y 533.567,Z 509.123,A -85,B 0,C 180,E1 21035.298,E2 21035.298} C_VEL
LIN {X 0,Y 539.82,Z 517.242,A -85,B 0,C 180,E1 21033.635,E2 21033.635} C_VEL
LIN {X 0,Y 550.215,Z 531.564,A -85,B 0,C 180,E1 21031.122,E2 21031.122} C_VEL
LIN {X 0,Y 558.03,Z 543.029,A -85,B 0,C 180,E1 21029.397,E2 21029.397} C_VEL
LIN {X 0,Y 546.574,Z 760.751,A -85,B 0,C 180,E1 21026.066,E2 21026.066} C_VEL
LIN {X 0,Y 540.461,Z 879.11,A -85,B 0,C 180,E1 21024.249,E2 21024.249} C_VEL
LIN {X 0,Y 538.065,Z 905.803,A -85,B 0,C 180,E1 21023.732,E2 21023.732} C_VEL
LIN {X 0,Y 534.612,Z 932.558,A -85,B 0,C 180,E1 21023.019,E2 21023.019} C_VEL
LIN {X 0,Y 531.403,Z 953.337,A -85,B 0,C 180,E1 21022.331,E2 21022.331} C_VEL
LIN {X 0,Y 527.859,Z 973.244,A -85,B 0,C 180,E1 21021.548,E2 21021.548} C_VEL
LIN {X 0,Y 523.809,Z 993.444,A -85,B 0,C 180,E1 21020.621,E2 21020.621} C_VEL
LIN {X 0,Y 518.999,Z 1015.197,A -85,B 0,C 180,E1 21019.455,E2 21019.455} C_VEL
LIN {X 0,Y 512.596,Z 1040.896,A -85,B 0,C 180,E1 21017.826,E2 21017.826} C_VEL
LIN {X 0,Y 507.343,Z 1060.328,A -85,B 0,C 180,E1 21016.386,E2 21016.386} C_VEL
LIN {X 0,Y 502.421,Z 1077.572,A -85,B 0,C 180,E1 21014.94,E2 21014.94} C_VEL
LIN {X 0,Y 497.336,Z 1094.626,A -85,B 0,C 180,E1 21013.333,E2 21013.333} C_VEL
LIN {X 0,Y 491.496,Z 1113.667,A -85,B 0,C 180,E1 21011.302,E2 21011.302} C_VEL
LIN {X 0,Y 485.029,Z 1133.891,A -85,B 0,C 180,E1 21008.797,E2 21008.797} C_VEL
LIN {X 0,Y 480.252,Z 1148.826,A -85,B 0,C 180,E1 21006.684,E2 21006.684} C_VEL
LIN {X 0,Y 475.729,Z 1163.074,A -85,B 0,C 180,E1 21004.42,E2 21004.42} C_VEL
LIN {X 0,Y 471.727,Z 1176.083,A -85,B 0,C 180,E1 21002.093,E2 21002.093} C_VEL
LIN {X 0,Y 469.603,Z 1180.357,A -85,B 0,C 180,E1 21001.346,E2 21001.346} C_VEL
LIN {X 0,Y 460.624,Z 1191.646,A -85,B 0,C 180,E1 20999.418,E2 20999.418} C_VEL
LIN {X 0,Y 458.965,Z 1194.835,A -85,B 0,C 180,E1 20998.724,E2 20998.724} C_VEL
LIN {X 0,Y 456.017,Z 1205.24,A -85,B 0,C 180,E1 20996.142,E2 20996.142} C_VEL
LIN {X 0,Y 453.242,Z 1216.035,A -85,B 0,C 180,E1 20993.082,E2 20993.082} C_VEL
LIN {X 0,Y 450.912,Z 1226.408,A -85,B 0,C 180,E1 20989.555,E2 20989.555} C_VEL
LIN {X 0,Y 449.673,Z 1233.234,A -85,B 0,C 180,E1 20986.795,E2 20986.795} C_VEL
LIN {X 0,Y 448.849,Z 1238.708,A -85,B 0,C 180,E1 20984.178,E2 20984.178} C_VEL
LIN {X 0,Y 448.343,Z 1243.412,A -85,B 0,C 180,E1 20981.442,E2 20981.442} C_VEL
LIN {X 0,Y 448.071,Z 1247.152,A -85,B 0,C 180,E1 20978.668,E2 20978.668} C_VEL
LIN {X 0,Y 447.946,Z 1250.096,A -85,B 0,C 180,E1 20975.63,E2 20975.63} C_VEL
LIN {X 0,Y 447.914,Z 1251.936,A -85,B 0,C 180,E1 20972.169,E2 20972.169} C_VEL
LIN {X 0,Y 447.871,Z 1252.192,A -85,B 0,C 180,E1 20969.227,E2 20969.227} C_VEL
LIN {X 0,Y 447.918,Z 1251.44,A -85,B 0,C 180,E1 20966.539,E2 20966.539} C_VEL
LIN {X 0,Y 447.963,Z 1249.723,A -85,B 0,C 180,E1 20963.844,E2 20963.844} C_VEL
LIN {X 0,Y 448.076,Z 1247.028,A -85,B 0,C 180,E1 20961.137,E2 20961.137} C_VEL
LIN {X 0,Y 448.345,Z 1243.333,A -85,B 0,C 180,E1 20958.416,E2 20958.416} C_VEL
LIN {X 0,Y 448.835,Z 1238.855,A -85,B 0,C 180,E1 20955.81,E2 20955.81} C_VEL
LIN {X 0,Y 449.689,Z 1233.114,A -85,B 0,C 180,E1 20953.06,E2 20953.06} C_VEL
LIN {X 0,Y 451.09,Z 1225.554,A -85,B 0,C 180,E1 20950.026,E2 20950.026} C_VEL
LIN {X 0,Y 453.511,Z 1214.838,A -85,B 0,C 180,E1 20946.475,E2 20946.475} C_VEL
LIN {X 0,Y 456.073,Z 1205.009,A -85,B 0,C 180,E1 20943.709,E2 20943.709} C_VEL
LIN {X 0,Y 459.092,Z 1194.381,A -85,B 0,C 180,E1 20941.08,E2 20941.08} C_VEL
LIN {X 0,Y 462.77,Z 1182.406,A -85,B 0,C 180,E1 20938.47,E2 20938.47} C_VEL
LIN {X 0,Y 468.264,Z 1165.263,A -85,B 0,C 180,E1 20935.236,E2 20935.236} C_VEL
LIN {X 0,Y 473.185,Z 1150.365,A -85,B 0,C 180,E1 20932.814,E2 20932.814} C_VEL
LIN {X 0,Y 478.121,Z 1135.544,A -85,B 0,C 180,E1 20930.675,E2 20930.675} C_VEL
LIN {X 0,Y 484.091,Z 1117.645,A -85,B 0,C 180,E1 20928.393,E2 20928.393} C_VEL
LIN {X 0,Y 490.868,Z 1096.571,A -85,B 0,C 180,E1 20926.081,E2 20926.081} C_VEL
LIN {X 0,Y 496.259,Z 1079.161,A -85,B 0,C 180,E1 20924.413,E2 20924.413} C_VEL
LIN {X 0,Y 501.365,Z 1061.935,A -85,B 0,C 180,E1 20922.948,E2 20922.948} C_VEL
LIN {X 0,Y 506.514,Z 1043.551,A -85,B 0,C 180,E1 20921.564,E2 20921.564} C_VEL
LIN {X 0,Y 512.153,Z 1022.027,A -85,B 0,C 180,E1 20920.148,E2 20920.148} C_VEL
LIN {X 0,Y 518.279,Z 995.882,A -85,B 0,C 180,E1 20918.701,E2 20918.701} C_VEL
LIN {X 0,Y 522.681,Z 974.7,A -85,B 0,C 180,E1 20917.715,E2 20917.715} C_VEL
LIN {X 0,Y 526.454,Z 954.225,A -85,B 0,C 180,E1 20916.904,E2 20916.904} C_VEL
LIN {X 0,Y 529.805,Z 933.197,A -85,B 0,C 180,E1 20916.204,E2 20916.204} C_VEL
LIN {X 0,Y 533.349,Z 906.604,A -85,B 0,C 180,E1 20915.492,E2 20915.492} C_VEL
LIN {X 0,Y 535.853,Z 879.629,A -85,B 0,C 180,E1 20914.966,E2 20914.966} C_VEL
LIN {X 0,Y 541.434,Z 775.606,A -85,B 0,C 180,E1 20913.361,E2 20913.361} C_VEL
LIN {X 0,Y 553.382,Z 555.487,A -85,B 0,C 180,E1 20909.984,E2 20909.984} C_VEL
LIN {X 0,Y 553.713,Z 547.339,A -85,B 0,C 180,E1 20909.835,E2 20909.835} C_VEL
LIN {X 0,Y 543.411,Z 532.467,A -85,B 0,C 180,E1 20907.447,E2 20907.447} C_VEL
LIN {X 0,Y 534.244,Z 519.961,A -85,B 0,C 180,E1 20905.082,E2 20905.082} C_VEL
LIN {X 0,Y 527.609,Z 511.31,A -85,B 0,C 180,E1 20903.186,E2 20903.186} C_VEL
LIN {X 0,Y 523.866,Z 506.512,A -85,B 0,C 180,E1 20902.028,E2 20902.028} C_VEL
LIN {X 0,Y 520.229,Z 501.917,A -85,B 0,C 180,E1 20900.829,E2 20900.829} C_VEL
LIN {X 0,Y 515.927,Z 496.517,A -85,B 0,C 180,E1 20899.295,E2 20899.295} C_VEL
LIN {X 0,Y 511.551,Z 491.115,A -85,B 0,C 180,E1 20897.577,E2 20897.577} C_VEL
LIN {X 0,Y 507.922,Z 486.789,A -85,B 0,C 180,E1 20895.998,E2 20895.998} C_VEL
LIN {X 0,Y 506.759,Z 485.314,A -85,B 0,C 180,E1 20895.448,E2 20895.448} C_VEL
LIN {X 0,Y 503.45,Z 481.745,A -85,B 0,C 180,E1 20893.788,E2 20893.788} C_VEL
LIN {X 0,Y 502.119,Z 479.52,A -85,B 0,C 180,E1 20893.004,E2 20893.004} C_VEL
LIN {X 0,Y 498.785,Z 476.669,A -85,B 0,C 180,E1 20890.979,E2 20890.979} C_VEL
LIN {X 0,Y 496.782,Z 473.181,A -85,B 0,C 180,E1 20889.383,E2 20889.383} C_VEL
LIN {X 0,Y 492.973,Z 470.119,A -85,B 0,C 180,E1 20885.587,E2 20885.587} C_VEL
LIN {X 0,Y 491.721,Z 466.726,A -85,B 0,C 180,E1 20882.797,E2 20882.797} C_VEL
LIN {X 0,Y 491.82,Z 466.926,A -85,B 0,C 180,E1 20877.32,E2 20877.32} C_VEL
LIN {X 0,Y 493.729,Z 471.119,A -85,B 0,C 180,E1 20873.838,E2 20873.838} C_VEL
LIN {X 0,Y 497.144,Z 473.628,A -85,B 0,C 180,E1 20870.741,E2 20870.741} C_VEL
LIN {X 0,Y 499.374,Z 477.416,A -85,B 0,C 180,E1 20869.034,E2 20869.034} C_VEL
LIN {X 0,Y 502.419,Z 479.927,A -85,B 0,C 180,E1 20867.238,E2 20867.238} C_VEL
LIN {X 0,Y 505.371,Z 484.125,A -85,B 0,C 180,E1 20865.623,E2 20865.623} C_VEL
LIN {X 0,Y 507.48,Z 486.085,A -85,B 0,C 180,E1 20864.633,E2 20864.633} C_VEL
LIN {X 0,Y 510.892,Z 490.549,A -85,B 0,C 180,E1 20863.104,E2 20863.104} C_VEL
LIN {X 0,Y 513.547,Z 493.762,A -85,B 0,C 180,E1 20862.025,E2 20862.025} C_VEL
LIN {X 0,Y 519.841,Z 502.367,A -85,B 0,C 180,E1 20859.685,E2 20859.685} C_VEL
LIN {X 0,Y 526.031,Z 510.844,A -85,B 0,C 180,E1 20857.656,E2 20857.656} C_VEL
LIN {X 0,Y 534.518,Z 523.28,A -85,B 0,C 180,E1 20855.168,E2 20855.168} C_VEL
LIN {X 0,Y 542.132,Z 534.844,A -85,B 0,C 180,E1 20853.166,E2 20853.166} C_VEL
LIN {X 0,Y 550.983,Z 548.779,A -85,B 0,C 180,E1 20851.048,E2 20851.048} C_VEL
LIN {X 0,Y 553.886,Z 553.857,A -85,B 0,C 180,E1 20850.384,E2 20850.384} C_VEL
LIN {X 0,Y 542.412,Z 766.437,A -85,B 0,C 180,E1 20847.116,E2 20847.116} C_VEL
LIN {X 0,Y 535.4,Z 899.309,A -85,B 0,C 180,E1 20845.071,E2 20845.071} C_VEL
LIN {X 0,Y 532.845,Z 926.508,A -85,B 0,C 180,E1 20844.555,E2 20844.555} C_VEL
LIN {X 0,Y 529.2,Z 953.17,A -85,B 0,C 180,E1 20843.869,E2 20843.869} C_VEL
LIN {X 0,Y 525.641,Z 974.956,A -85,B 0,C 180,E1 20843.169,E2 20843.169} C_VEL
LIN {X 0,Y 521.917,Z 995.009,A -85,B 0,C 180,E1 20842.394,E2 20842.394} C_VEL
LIN {X 0,Y 517.661,Z 1015.405,A -85,B 0,C 180,E1 20841.474,E2 20841.474} C_VEL
LIN {X 0,Y 512.414,Z 1038.445,A -85,B 0,C 180,E1 20840.252,E2 20840.252} C_VEL
LIN {X 0,Y 506.146,Z 1062.931,A -85,B 0,C 180,E1 20838.714,E2 20838.714} C_VEL
LIN {X 0,Y 500.771,Z 1082.438,A -85,B 0,C 180,E1 20837.293,E2 20837.293} C_VEL
LIN {X 0,Y 495.617,Z 1100.203,A -85,B 0,C 180,E1 20835.829,E2 20835.829} C_VEL
LIN {X 0,Y 490.243,Z 1118.048,A -85,B 0,C 180,E1 20834.169,E2 20834.169} C_VEL
LIN {X 0,Y 483.808,Z 1138.995,A -85,B 0,C 180,E1 20831.954,E2 20831.954} C_VEL
LIN {X 0,Y 477.551,Z 1158.583,A -85,B 0,C 180,E1 20829.536,E2 20829.536} C_VEL
LIN {X 0,Y 472.655,Z 1173.974,A -85,B 0,C 180,E1 20827.387,E2 20827.387} C_VEL
LIN {X 0,Y 468.294,Z 1187.909,A -85,B 0,C 180,E1 20825.209,E2 20825.209} C_VEL
LIN {X 0,Y 463.996,Z 1201.959,A -85,B 0,C 180,E1 20822.749,E2 20822.749} C_VEL
LIN {X 0,Y 459.137,Z 1218.811,A -85,B 0,C 180,E1 20819.345,E2 20819.345} C_VEL
LIN {X 0,Y 456.094,Z 1230.097,A -85,B 0,C 180,E1 20816.711,E2 20816.711} C_VEL
LIN {X 0,Y 453.667,Z 1240.101,A -85,B 0,C 180,E1 20814.068,E2 20814.068} C_VEL
LIN {X 0,Y 451.788,Z 1248.899,A -85,B 0,C 180,E1 20811.423,E2 20811.423} C_VEL
LIN {X 0,Y 450.155,Z 1257.638,A -85,B 0,C 180,E1 20808.391,E2 20808.391} C_VEL
LIN {X 0,Y 448.917,Z 1266.048,A -85,B 0,C 180,E1 20804.835,E2 20804.835} C_VEL
LIN {X 0,Y 448.375,Z 1271.457,A -85,B 0,C 180,E1 20801.975,E2 20801.975} C_VEL
LIN {X 0,Y 448.054,Z 1275.542,A -85,B 0,C 180,E1 20799.252,E2 20799.252} C_VEL
LIN {X 0,Y 447.963,Z 1278.57,A -85,B 0,C 180,E1 20796.542,E2 20796.542} C_VEL
LIN {X 0,Y 447.92,Z 1280.486,A -85,B 0,C 180,E1 20793.974,E2 20793.974} C_VEL
LIN {X 0,Y 447.902,Z 1281.466,A -85,B 0,C 180,E1 20791.413,E2 20791.413} C_VEL
LIN {X 0,Y 447.88,Z 1281.538,A -85,B 0,C 180,E1 20788.983,E2 20788.983} C_VEL
LIN {X 0,Y 447.917,Z 1280.702,A -85,B 0,C 180,E1 20786.422,E2 20786.422} C_VEL
LIN {X 0,Y 447.954,Z 1278.931,A -85,B 0,C 180,E1 20783.856,E2 20783.856} C_VEL
LIN {X 0,Y 448.052,Z 1276.05,A -85,B 0,C 180,E1 20781.149,E2 20781.149} C_VEL
LIN {X 0,Y 448.294,Z 1272.327,A -85,B 0,C 180,E1 20778.557,E2 20778.557} C_VEL
LIN {X 0,Y 448.742,Z 1267.619,A -85,B 0,C 180,E1 20775.951,E2 20775.951} C_VEL
LIN {X 0,Y 449.489,Z 1261.9,A -85,B 0,C 180,E1 20773.331,E2 20773.331} C_VEL
LIN {X 0,Y 450.649,Z 1254.749,A -85,B 0,C 180,E1 20770.559,E2 20770.559} C_VEL
LIN {X 0,Y 452.657,Z 1244.786,A -85,B 0,C 180,E1 20767.267,E2 20767.267} C_VEL
LIN {X 0,Y 455.442,Z 1232.784,A -85,B 0,C 180,E1 20763.963,E2 20763.963} C_VEL
LIN {X 0,Y 458.351,Z 1221.596,A -85,B 0,C 180,E1 20761.278,E2 20761.278} C_VEL
LIN {X 0,Y 461.791,Z 1209.442,A -85,B 0,C 180,E1 20758.699,E2 20758.699} C_VEL
LIN {X 0,Y 466.382,Z 1194.174,A -85,B 0,C 180,E1 20755.835,E2 20755.835} C_VEL
LIN {X 0,Y 471.816,Z 1176.62,A -85,B 0,C 180,E1 20753.006,E2 20753.006} C_VEL
LIN {X 0,Y 476.69,Z 1161.219,A -85,B 0,C 180,E1 20750.817,E2 20750.817} C_VEL
LIN {X 0,Y 481.693,Z 1145.459,A -85,B 0,C 180,E1 20748.819,E2 20748.819} C_VEL
LIN {X 0,Y 487.452,Z 1127.209,A -85,B 0,C 180,E1 20746.765,E2 20746.765} C_VEL
LIN {X 0,Y 494.387,Z 1104.397,A -85,B 0,C 180,E1 20744.546,E2 20744.546} C_VEL
LIN {X 0,Y 499.891,Z 1085.483,A -85,B 0,C 180,E1 20742.95,E2 20742.95} C_VEL
LIN {X 0,Y 504.824,Z 1067.68,A -85,B 0,C 180,E1 20741.62,E2 20741.62} C_VEL
LIN {X 0,Y 509.759,Z 1048.735,A -85,B 0,C 180,E1 20740.367,E2 20740.367} C_VEL
LIN {X 0,Y 514.853,Z 1027.757,A -85,B 0,C 180,E1 20739.159,E2 20739.159} C_VEL
LIN {X 0,Y 520.605,Z 1001.582,A -85,B 0,C 180,E1 20737.885,E2 20737.885} C_VEL
LIN {X 0,Y 525.063,Z 978.051,A -85,B 0,C 180,E1 20736.946,E2 20736.946} C_VEL
LIN {X 0,Y 528.659,Z 956.397,A -85,B 0,C 180,E1 20736.23,E2 20736.23} C_VEL
LIN {X 0,Y 531.655,Z 935.103,A -85,B 0,C 180,E1 20735.652,E2 20735.652} C_VEL
LIN {X 0,Y 534.416,Z 910.896,A -85,B 0,C 180,E1 20735.136,E2 20735.136} C_VEL
LIN {X 0,Y 536.808,Z 874.633,A -85,B 0,C 180,E1 20734.539,E2 20734.539} C_VEL
LIN {X 0,Y 548.26,Z 655.134,A -85,B 0,C 180,E1 20731.182,E2 20731.182} C_VEL
LIN {X 0,Y 553.734,Z 553.451,A -85,B 0,C 180,E1 20729.595,E2 20729.595} C_VEL
LIN {X 0,Y 544.015,Z 537.785,A -85,B 0,C 180,E1 20727.325,E2 20727.325} C_VEL
LIN {X 0,Y 534.968,Z 524.021,A -85,B 0,C 180,E1 20724.987,E2 20724.987} C_VEL
LIN {X 0,Y 526.986,Z 512.416,A -85,B 0,C 180,E1 20722.684,E2 20722.684} C_VEL
LIN {X 0,Y 521.323,Z 504.515,A -85,B 0,C 180,E1 20720.871,E2 20720.871} C_VEL
LIN {X 0,Y 517.474,Z 499.256,A -85,B 0,C 180,E1 20719.529,E2 20719.529} C_VEL
LIN {X 0,Y 512.727,Z 492.794,A -85,B 0,C 180,E1 20717.711,E2 20717.711} C_VEL
LIN {X 0,Y 510.604,Z 490.349,A -85,B 0,C 180,E1 20716.847,E2 20716.847} C_VEL
LIN {X 0,Y 507.266,Z 485.833,A -85,B 0,C 180,E1 20715.345,E2 20715.345} C_VEL
LIN {X 0,Y 503.39,Z 481.76,A -85,B 0,C 180,E1 20713.438,E2 20713.438} C_VEL
LIN {X 0,Y 502.046,Z 479.529,A -85,B 0,C 180,E1 20712.655,E2 20712.655} C_VEL
LIN {X 0,Y 498.762,Z 476.774,A -85,B 0,C 180,E1 20710.687,E2 20710.687} C_VEL
LIN {X 0,Y 496.809,Z 473.21,A -85,B 0,C 180,E1 20709.149,E2 20709.149} C_VEL
LIN {X 0,Y 493.038,Z 470.409,A -85,B 0,C 180,E1 20705.586,E2 20705.586} C_VEL
LIN {X 0,Y 491.577,Z 466.721,A -85,B 0,C 180,E1 20702.681,E2 20702.681} C_VEL
LIN {X 0,Y 491.703,Z 466.86,A -85,B 0,C 180,E1 20696.502,E2 20696.502} C_VEL
LIN {X 0,Y 493.106,Z 470.41,A -85,B 0,C 180,E1 20693.83,E2 20693.83} C_VEL
LIN {X 0,Y 496.756,Z 473.203,A -85,B 0,C 180,E1 20690.383,E2 20690.383} C_VEL
LIN {X 0,Y 499.299,Z 477.389,A -85,B 0,C 180,E1 20688.448,E2 20688.448} C_VEL
LIN {X 0,Y 502.372,Z 479.952,A -85,B 0,C 180,E1 20686.651,E2 20686.651} C_VEL
LIN {X 0,Y 505.238,Z 484.077,A -85,B 0,C 180,E1 20685.091,E2 20685.091} C_VEL
LIN {X 0,Y 507.475,Z 486.193,A -85,B 0,C 180,E1 20684.046,E2 20684.046} C_VEL
LIN {X 0,Y 510.925,Z 490.594,A -85,B 0,C 180,E1 20682.518,E2 20682.518} C_VEL
LIN {X 0,Y 512.531,Z 492.332,A -85,B 0,C 180,E1 20681.87,E2 20681.87} C_VEL
LIN {X 0,Y 517.386,Z 498.392,A -85,B 0,C 180,E1 20680.026,E2 20680.026} C_VEL
LIN {X 0,Y 522.295,Z 504.576,A -85,B 0,C 180,E1 20678.346,E2 20678.346} C_VEL
LIN {X 0,Y 526.644,Z 510.144,A -85,B 0,C 180,E1 20676.976,E2 20676.976} C_VEL
LIN {X 0,Y 534.056,Z 519.726,A -85,B 0,C 180,E1 20674.849,E2 20674.849} C_VEL
LIN {X 0,Y 544.325,Z 533.807,A -85,B 0,C 180,E1 20672.217,E2 20672.217} C_VEL
LIN {X 0,Y 553.758,Z 547.551,A -85,B 0,C 180,E1 20670.045,E2 20670.045} C_VEL
LIN {X 0,Y 541.866,Z 766.348,A -85,B 0,C 180,E1 20666.687,E2 20666.687} C_VEL
LIN {X 0,Y 535.821,Z 879.423,A -85,B 0,C 180,E1 20664.944,E2 20664.944} C_VEL
LIN {X 0,Y 533.331,Z 906.392,A -85,B 0,C 180,E1 20664.419,E2 20664.419} C_VEL
LIN {X 0,Y 529.802,Z 932.942,A -85,B 0,C 180,E1 20663.71,E2 20663.71} C_VEL
LIN {X 0,Y 526.519,Z 953.612,A -85,B 0,C 180,E1 20663.025,E2 20663.025} C_VEL
LIN {X 0,Y 522.875,Z 973.517,A -85,B 0,C 180,E1 20662.242,E2 20662.242} C_VEL
LIN {X 0,Y 518.708,Z 993.718,A -85,B 0,C 180,E1 20661.312,E2 20661.312} C_VEL
LIN {X 0,Y 513.754,Z 1015.471,A -85,B 0,C 180,E1 20660.144,E2 20660.144} C_VEL
LIN {X 0,Y 507.151,Z 1041.169,A -85,B 0,C 180,E1 20658.51,E2 20658.51} C_VEL
LIN {X 0,Y 501.969,Z 1059.768,A -85,B 0,C 180,E1 20657.13,E2 20657.13} C_VEL
LIN {X 0,Y 496.83,Z 1077.186,A -85,B 0,C 180,E1 20655.67,E2 20655.67} C_VEL
LIN {X 0,Y 491.581,Z 1094.171,A -85,B 0,C 180,E1 20654.067,E2 20654.067} C_VEL
LIN {X 0,Y 486.035,Z 1111.55,A -85,B 0,C 180,E1 20652.217,E2 20652.217} C_VEL
LIN {X 0,Y 479.15,Z 1132.528,A -85,B 0,C 180,E1 20649.643,E2 20649.643} C_VEL
LIN {X 0,Y 473.883,Z 1148.271,A -85,B 0,C 180,E1 20647.412,E2 20647.412} C_VEL
LIN {X 0,Y 469.385,Z 1161.836,A -85,B 0,C 180,E1 20645.251,E2 20645.251} C_VEL
LIN {X 0,Y 465.166,Z 1174.788,A -85,B 0,C 180,E1 20642.936,E2 20642.936} C_VEL
LIN {X 0,Y 460.949,Z 1188.302,A -85,B 0,C 180,E1 20640.207,E2 20640.207} C_VEL
LIN {X 0,Y 458.965,Z 1194.835,A -85,B 0,C 180,E1 20638.724,E2 20638.724} C_VEL
LIN {X 0,Y 456.983,Z 1198.635,A -85,B 0,C 180,E1 20637.909,E2 20637.909} C_VEL
LIN {X 0,Y 448.477,Z 1208.438,A -85,B 0,C 180,E1 20635.782,E2 20635.782} C_VEL
LIN {X 0,Y 446.979,Z 1211.193,A -85,B 0,C 180,E1 20635.03,E2 20635.03} C_VEL
LIN {X 0,Y 444.631,Z 1220.276,A -85,B 0,C 180,E1 20632.19,E2 20632.19} C_VEL
LIN {X 0,Y 442.864,Z 1228.056,A -85,B 0,C 180,E1 20629.376,E2 20629.376} C_VEL
LIN {X 0,Y 441.622,Z 1234.684,A -85,B 0,C 180,E1 20626.568,E2 20626.568} C_VEL
LIN {X 0,Y 440.683,Z 1241.202,A -85,B 0,C 180,E1 20623.241,E2 20623.241} C_VEL
LIN {X 0,Y 440.136,Z 1246.273,A -85,B 0,C 180,E1 20619.803,E2 20619.803} C_VEL
LIN {X 0,Y 439.985,Z 1249.479,A -85,B 0,C 180,E1 20616.78,E2 20616.78} C_VEL
LIN {X 0,Y 439.928,Z 1251.398,A -85,B 0,C 180,E1 20614.034,E2 20614.034} C_VEL
LIN {X 0,Y 439.91,Z 1252.329,A -85,B 0,C 180,E1 20611.427,E2 20611.427} C_VEL
LIN {X 0,Y 439.891,Z 1252.387,A -85,B 0,C 180,E1 20608.822,E2 20608.822} C_VEL
LIN {X 0,Y 439.929,Z 1251.555,A -85,B 0,C 180,E1 20606.186,E2 20606.186} C_VEL
LIN {X 0,Y 439.98,Z 1249.766,A -85,B 0,C 180,E1 20603.47,E2 20603.47} C_VEL
LIN {X 0,Y 440.092,Z 1246.984,A -85,B 0,C 180,E1 20600.711,E2 20600.711} C_VEL
LIN {X 0,Y 440.418,Z 1243.397,A -85,B 0,C 180,E1 20598.072,E2 20598.072} C_VEL
LIN {X 0,Y 440.946,Z 1238.875,A -85,B 0,C 180,E1 20595.416,E2 20595.416} C_VEL
LIN {X 0,Y 441.904,Z 1233.086,A -85,B 0,C 180,E1 20592.617,E2 20592.617} C_VEL
LIN {X 0,Y 443.677,Z 1224.45,A -85,B 0,C 180,E1 20589.136,E2 20589.136} C_VEL
LIN {X 0,Y 446.143,Z 1214.211,A -85,B 0,C 180,E1 20585.782,E2 20585.782} C_VEL
LIN {X 0,Y 448.754,Z 1204.776,A -85,B 0,C 180,E1 20583.103,E2 20583.103} C_VEL
LIN {X 0,Y 451.812,Z 1194.652,A -85,B 0,C 180,E1 20580.569,E2 20580.569} C_VEL
LIN {X 0,Y 455.771,Z 1182.424,A -85,B 0,C 180,E1 20577.868,E2 20577.868} C_VEL
LIN {X 0,Y 461.435,Z 1165.534,A -85,B 0,C 180,E1 20574.646,E2 20574.646} C_VEL
LIN {X 0,Y 466.352,Z 1151.28,A -85,B 0,C 180,E1 20572.295,E2 20572.295} C_VEL
LIN {X 0,Y 471.56,Z 1136.269,A -85,B 0,C 180,E1 20570.098,E2 20570.098} C_VEL
LIN {X 0,Y 477.223,Z 1119.867,A -85,B 0,C 180,E1 20567.973,E2 20567.973} C_VEL
LIN {X 0,Y 484.576,Z 1098.013,A -85,B 0,C 180,E1 20565.522,E2 20565.522} C_VEL
LIN {X 0,Y 490.328,Z 1080.087,A -85,B 0,C 180,E1 20563.785,E2 20563.785} C_VEL
LIN {X 0,Y 495.596,Z 1062.926,A -85,B 0,C 180,E1 20562.313,E2 20562.313} C_VEL
LIN {X 0,Y 500.672,Z 1045.422,A -85,B 0,C 180,E1 20560.979,E2 20560.979} C_VEL
LIN {X 0,Y 505.744,Z 1026.752,A -85,B 0,C 180,E1 20559.725,E2 20559.725} C_VEL
LIN {X 0,Y 511.288,Z 1004.7,A -85,B 0,C 180,E1 20558.439,E2 20558.439} C_VEL
LIN {X 0,Y 517.026,Z 978.784,A -85,B 0,C 180,E1 20557.173,E2 20557.173} C_VEL
LIN {X 0,Y 521.265,Z 956.687,A -85,B 0,C 180,E1 20556.277,E2 20556.277} C_VEL
LIN {X 0,Y 524.712,Z 935.952,A -85,B 0,C 180,E1 20555.573,E2 20555.573} C_VEL
LIN {X 0,Y 527.752,Z 914.278,A -85,B 0,C 180,E1 20554.969,E2 20554.969} C_VEL
LIN {X 0,Y 530.559,Z 889.197,A -85,B 0,C 180,E1 20554.42,E2 20554.42} C_VEL
LIN {X 0,Y 533.015,Z 851.746,A -85,B 0,C 180,E1 20553.81,E2 20553.81} C_VEL
LIN {X 0,Y 545.113,Z 630.789,A -85,B 0,C 180,E1 20550.418,E2 20550.418} C_VEL
LIN {X 0,Y 549.542,Z 552.026,A -85,B 0,C 180,E1 20549.185,E2 20549.185} C_VEL
LIN {X 0,Y 540.248,Z 538.562,A -85,B 0,C 180,E1 20546.965,E2 20546.965} C_VEL
LIN {X 0,Y 531.007,Z 525.674,A -85,B 0,C 180,E1 20544.503,E2 20544.503} C_VEL
LIN {X 0,Y 522.57,Z 514.632,A -85,B 0,C 180,E1 20541.967,E2 20541.967} C_VEL
LIN {X 0,Y 518.178,Z 509.123,A -85,B 0,C 180,E1 20540.501,E2 20540.501} C_VEL
LIN {X 0,Y 514.094,Z 503.922,A -85,B 0,C 180,E1 20539.013,E2 20539.013} C_VEL
LIN {X 0,Y 509.923,Z 498.69,A -85,B 0,C 180,E1 20537.341,E2 20537.341} C_VEL
LIN {X 0,Y 506.243,Z 494.153,A -85,B 0,C 180,E1 20535.7,E2 20535.7} C_VEL
LIN {X 0,Y 505.087,Z 492.837,A -85,B 0,C 180,E1 20535.148,E2 20535.148} C_VEL
LIN {X 0,Y 501.776,Z 488.98,A -85,B 0,C 180,E1 20533.424,E2 20533.424} C_VEL
LIN {X 0,Y 500.75,Z 487.287,A -85,B 0,C 180,E1 20532.806,E2 20532.806} C_VEL
LIN {X 0,Y 497.409,Z 484.254,A -85,B 0,C 180,E1 20530.716,E2 20530.716} C_VEL
LIN {X 0,Y 495.667,Z 481.075,A -85,B 0,C 180,E1 20529.287,E2 20529.287} C_VEL
LIN {X 0,Y 491.918,Z 477.998,A -85,B 0,C 180,E1 20525.482,E2 20525.482} C_VEL
LIN {X 0,Y 490.747,Z 474.667,A -85,B 0,C 180,E1 20522.803,E2 20522.803} C_VEL
LIN {X 0,Y 490.803,Z 474.815,A -85,B 0,C 180,E1 20517.431,E2 20517.431} C_VEL
LIN {X 0,Y 492.754,Z 479.104,A -85,B 0,C 180,E1 20513.826,E2 20513.826} C_VEL
LIN {X 0,Y 495.947,Z 481.484,A -85,B 0,C 180,E1 20510.894,E2 20510.894} C_VEL
LIN {X 0,Y 498.229,Z 485.309,A -85,B 0,C 180,E1 20509.126,E2 20509.126} C_VEL
LIN {X 0,Y 501.137,Z 487.829,A -85,B 0,C 180,E1 20507.38,E2 20507.38} C_VEL
LIN {X 0,Y 504.291,Z 492.148,A -85,B 0,C 180,E1 20505.65,E2 20505.65} C_VEL
LIN {X 0,Y 506.029,Z 493.834,A -85,B 0,C 180,E1 20504.822,E2 20504.822} C_VEL
LIN {X 0,Y 509.535,Z 498.36,A -85,B 0,C 180,E1 20503.234,E2 20503.234} C_VEL
LIN {X 0,Y 514.058,Z 504.342,A -85,B 0,C 180,E1 20501.398,E2 20501.398} C_VEL
LIN {X 0,Y 518.467,Z 510.501,A -85,B 0,C 180,E1 20499.776,E2 20499.776} C_VEL
LIN {X 0,Y 523.966,Z 518.113,A -85,B 0,C 180,E1 20497.947,E2 20497.947} C_VEL
LIN {X 0,Y 533.521,Z 532.23,A -85,B 0,C 180,E1 20495.118,E2 20495.118} C_VEL
LIN {X 0,Y 542.876,Z 546.902,A -85,B 0,C 180,E1 20492.672,E2 20492.672} C_VEL
LIN {X 0,Y 549.68,Z 558.196,A -85,B 0,C 180,E1 20491.044,E2 20491.044} C_VEL
LIN {X 0,Y 537.83,Z 770.855,A -85,B 0,C 180,E1 20487.764,E2 20487.764} C_VEL
LIN {X 0,Y 530.824,Z 899.171,A -85,B 0,C 180,E1 20485.782,E2 20485.782} C_VEL
LIN {X 0,Y 528.171,Z 926.609,A -85,B 0,C 180,E1 20485.26,E2 20485.26} C_VEL
LIN {X 0,Y 524.434,Z 953.141,A -85,B 0,C 180,E1 20484.577,E2 20484.577} C_VEL
LIN {X 0,Y 520.832,Z 974.598,A -85,B 0,C 180,E1 20483.887,E2 20483.887} C_VEL
LIN {X 0,Y 516.981,Z 994.748,A -85,B 0,C 180,E1 20483.11,E2 20483.11} C_VEL
LIN {X 0,Y 512.604,Z 1015.142,A -85,B 0,C 180,E1 20482.189,E2 20482.189} C_VEL
LIN {X 0,Y 507.19,Z 1038.18,A -85,B 0,C 180,E1 20480.967,E2 20480.967} C_VEL
LIN {X 0,Y 500.791,Z 1062.417,A -85,B 0,C 180,E1 20479.443,E2 20479.443} C_VEL
LIN {X 0,Y 495.164,Z 1082.169,A -85,B 0,C 180,E1 20478.001,E2 20478.001} C_VEL
LIN {X 0,Y 489.627,Z 1100.607,A -85,B 0,C 180,E1 20476.47,E2 20476.47} C_VEL
LIN {X 0,Y 483.826,Z 1119.193,A -85,B 0,C 180,E1 20474.719,E2 20474.719} C_VEL
LIN {X 0,Y 476.635,Z 1141.534,A -85,B 0,C 180,E1 20472.293,E2 20472.293} C_VEL
LIN {X 0,Y 470.759,Z 1159.248,A -85,B 0,C 180,E1 20470.063,E2 20470.063} C_VEL
LIN {X 0,Y 465.964,Z 1173.699,A -85,B 0,C 180,E1 20468.019,E2 20468.019} C_VEL
LIN {X 0,Y 461.414,Z 1187.634,A -85,B 0,C 180,E1 20465.814,E2 20465.814} C_VEL
LIN {X 0,Y 456.826,Z 1201.977,A -85,B 0,C 180,E1 20463.268,E2 20463.268} C_VEL
LIN {X 0,Y 451.806,Z 1218.535,A -85,B 0,C 180,E1 20459.869,E2 20459.869} C_VEL
LIN {X 0,Y 448.595,Z 1229.821,A -85,B 0,C 180,E1 20457.194,E2 20457.194} C_VEL
LIN {X 0,Y 446.036,Z 1239.826,A -85,B 0,C 180,E1 20454.507,E2 20454.507} C_VEL
LIN {X 0,Y 443.953,Z 1249.04,A -85,B 0,C 180,E1 20451.682,E2 20451.682} C_VEL
LIN {X 0,Y 442.069,Z 1258.797,A -85,B 0,C 180,E1 20448.193,E2 20448.193} C_VEL
LIN {X 0,Y 440.92,Z 1266.279,A -85,B 0,C 180,E1 20444.853,E2 20444.853} C_VEL
LIN {X 0,Y 440.387,Z 1271.402,A -85,B 0,C 180,E1 20442.062,E2 20442.062} C_VEL
LIN {X 0,Y 440.061,Z 1275.276,A -85,B 0,C 180,E1 20439.421,E2 20439.421} C_VEL
LIN {X 0,Y 439.967,Z 1278.263,A -85,B 0,C 180,E1 20436.709,E2 20436.709} C_VEL
LIN {X 0,Y 439.923,Z 1280.223,A -85,B 0,C 180,E1 20434.046,E2 20434.046} C_VEL
LIN {X 0,Y 439.907,Z 1281.204,A -85,B 0,C 180,E1 20431.439,E2 20431.439} C_VEL
LIN {X 0,Y 439.885,Z 1281.275,A -85,B 0,C 180,E1 20428.964,E2 20428.964} C_VEL
LIN {X 0,Y 439.921,Z 1280.439,A -85,B 0,C 180,E1 20426.357,E2 20426.357} C_VEL
LIN {X 0,Y 439.96,Z 1278.667,A -85,B 0,C 180,E1 20423.744,E2 20423.744} C_VEL
LIN {X 0,Y 440.051,Z 1275.784,A -85,B 0,C 180,E1 20420.986,E2 20420.986} C_VEL
LIN {X 0,Y 440.322,Z 1272.06,A -85,B 0,C 180,E1 20418.347,E2 20418.347} C_VEL
LIN {X 0,Y 440.789,Z 1267.35,A -85,B 0,C 180,E1 20415.692,E2 20415.692} C_VEL
LIN {X 0,Y 441.601,Z 1261.63,A -85,B 0,C 180,E1 20413.024,E2 20413.024} C_VEL
LIN {X 0,Y 442.815,Z 1254.498,A -85,B 0,C 180,E1 20410.21,E2 20410.21} C_VEL
LIN {X 0,Y 444.757,Z 1245.342,A -85,B 0,C 180,E1 20407.12,E2 20407.12} C_VEL
LIN {X 0,Y 447.764,Z 1233.034,A -85,B 0,C 180,E1 20403.624,E2 20403.624} C_VEL
LIN {X 0,Y 450.778,Z 1222.009,A -85,B 0,C 180,E1 20400.921,E2 20400.921} C_VEL
LIN {X 0,Y 454.195,Z 1210.459,A -85,B 0,C 180,E1 20398.412,E2 20398.412} C_VEL
LIN {X 0,Y 458.238,Z 1197.463,A -85,B 0,C 180,E1 20395.899,E2 20395.899} C_VEL
LIN {X 0,Y 463.731,Z 1180.629,A -85,B 0,C 180,E1 20393.027,E2 20393.027} C_VEL
LIN {X 0,Y 469.527,Z 1162.925,A -85,B 0,C 180,E1 20390.435,E2 20390.435} C_VEL
LIN {X 0,Y 474.725,Z 1147.18,A -85,B 0,C 180,E1 20388.393,E2 20388.393} C_VEL
LIN {X 0,Y 480.06,Z 1130.867,A -85,B 0,C 180,E1 20386.509,E2 20386.509} C_VEL
LIN {X 0,Y 485.963,Z 1112.429,A -85,B 0,C 180,E1 20384.621,E2 20384.621} C_VEL
LIN {X 0,Y 493.404,Z 1088.175,A -85,B 0,C 180,E1 20382.48,E2 20382.48} C_VEL
LIN {X 0,Y 499.137,Z 1068.223,A -85,B 0,C 180,E1 20380.967,E2 20380.967} C_VEL
LIN {X 0,Y 504.22,Z 1049.368,A -85,B 0,C 180,E1 20379.71,E2 20379.71} C_VEL
LIN {X 0,Y 509.296,Z 1029.16,A -85,B 0,C 180,E1 20378.535,E2 20378.535} C_VEL
LIN {X 0,Y 514.601,Z 1006.134,A -85,B 0,C 180,E1 20377.386,E2 20377.386} C_VEL
LIN {X 0,Y 519.954,Z 979.264,A -85,B 0,C 180,E1 20376.284,E2 20376.284} C_VEL
LIN {X 0,Y 523.744,Z 957.211,A -85,B 0,C 180,E1 20375.548,E2 20375.548} C_VEL
LIN {X 0,Y 526.852,Z 935.867,A -85,B 0,C 180,E1 20374.965,E2 20374.965} C_VEL
LIN {X 0,Y 529.522,Z 913.386,A -85,B 0,C 180,E1 20374.479,E2 20374.479} C_VEL
LIN {X 0,Y 531.804,Z 883.573,A -85,B 0,C 180,E1 20373.966,E2 20373.966} C_VEL
LIN {X 0,Y 543.758,Z 661.539,A -85,B 0,C 180,E1 20370.559,E2 20370.559} C_VEL
LIN {X 0,Y 549.556,Z 557.961,A -85,B 0,C 180,E1 20368.945,E2 20368.945} C_VEL
LIN {X 0,Y 541.127,Z 544.23,A -85,B 0,C 180,E1 20366.918,E2 20366.918} C_VEL
LIN {X 0,Y 532.507,Z 530.907,A -85,B 0,C 180,E1 20364.636,E2 20364.636} C_VEL
LIN {X 0,Y 524.331,Z 518.814,A -85,B 0,C 180,E1 20362.214,E2 20362.214} C_VEL
LIN {X 0,Y 518.867,Z 511.149,A -85,B 0,C 180,E1 20360.414,E2 20360.414} C_VEL
LIN {X 0,Y 515.323,Z 506.244,A -85,B 0,C 180,E1 20359.142,E2 20359.142} C_VEL
LIN {X 0,Y 510.173,Z 499.058,A -85,B 0,C 180,E1 20357.097,E2 20357.097} C_VEL
LIN {X 0,Y 506.314,Z 494.448,A -85,B 0,C 180,E1 20355.404,E2 20355.404} C_VEL
LIN {X 0,Y 505.283,Z 493.055,A -85,B 0,C 180,E1 20354.907,E2 20354.907} C_VEL
LIN {X 0,Y 501.707,Z 489,A -85,B 0,C 180,E1 20353.074,E2 20353.074} C_VEL
LIN {X 0,Y 500.466,Z 487.187,A -85,B 0,C 180,E1 20352.344,E2 20352.344} C_VEL
LIN {X 0,Y 497.3,Z 484.238,A -85,B 0,C 180,E1 20350.367,E2 20350.367} C_VEL
LIN {X 0,Y 495.536,Z 481.043,A -85,B 0,C 180,E1 20348.938,E2 20348.938} C_VEL
LIN {X 0,Y 491.891,Z 478.159,A -85,B 0,C 180,E1 20345.365,E2 20345.365} C_VEL
LIN {X 0,Y 490.553,Z 474.656,A -85,B 0,C 180,E1 20342.57,E2 20342.57} C_VEL
LIN {X 0,Y 490.68,Z 474.751,A -85,B 0,C 180,E1 20336.612,E2 20336.612} C_VEL
LIN {X 0,Y 492.131,Z 478.398,A -85,B 0,C 180,E1 20333.818,E2 20333.818} C_VEL
LIN {X 0,Y 495.837,Z 481.465,A -85,B 0,C 180,E1 20330.306,E2 20330.306} C_VEL
LIN {X 0,Y 497.983,Z 485.094,A -85,B 0,C 180,E1 20328.652,E2 20328.652} C_VEL
LIN {X 0,Y 500.998,Z 487.684,A -85,B 0,C 180,E1 20326.849,E2 20326.849} C_VEL
LIN {X 0,Y 503.934,Z 491.883,A -85,B 0,C 180,E1 20325.228,E2 20325.228} C_VEL
LIN {X 0,Y 506.022,Z 493.94,A -85,B 0,C 180,E1 20324.235,E2 20324.235} C_VEL
LIN {X 0,Y 509.567,Z 498.405,A -85,B 0,C 180,E1 20322.647,E2 20322.647} C_VEL
LIN {X 0,Y 511.142,Z 500.294,A -85,B 0,C 180,E1 20321.996,E2 20321.996} C_VEL
LIN {X 0,Y 515.672,Z 505.967,A -85,B 0,C 180,E1 20320.253,E2 20320.253} C_VEL
LIN {X 0,Y 520.443,Z 512.05,A -85,B 0,C 180,E1 20318.59,E2 20318.59} C_VEL
LIN {X 0,Y 524.738,Z 517.63,A -85,B 0,C 180,E1 20317.214,E2 20317.214} C_VEL
LIN {X 0,Y 532.065,Z 527.259,A -85,B 0,C 180,E1 20315.075,E2 20315.075} C_VEL
LIN {X 0,Y 541.934,Z 540.985,A -85,B 0,C 180,E1 20312.502,E2 20312.502} C_VEL
LIN {X 0,Y 549.546,Z 552.259,A -85,B 0,C 180,E1 20310.7,E2 20310.7} C_VEL
LIN {X 0,Y 537.191,Z 772.528,A -85,B 0,C 180,E1 20307.31,E2 20307.31} C_VEL
LIN {X 0,Y 531.261,Z 879.744,A -85,B 0,C 180,E1 20305.65,E2 20305.65} C_VEL
LIN {X 0,Y 528.691,Z 906.818,A -85,B 0,C 180,E1 20305.122,E2 20305.122} C_VEL
LIN {X 0,Y 525.07,Z 933.326,A -85,B 0,C 180,E1 20304.414,E2 20304.414} C_VEL
LIN {X 0,Y 521.715,Z 953.886,A -85,B 0,C 180,E1 20303.731,E2 20303.731} C_VEL
LIN {X 0,Y 517.971,Z 973.791,A -85,B 0,C 180,E1 20302.948,E2 20302.948} C_VEL
LIN {X 0,Y 513.682,Z 993.992,A -85,B 0,C 180,E1 20302.018,E2 20302.018} C_VEL
LIN {X 0,Y 508.584,Z 1015.744,A -85,B 0,C 180,E1 20300.847,E2 20300.847} C_VEL
LIN {X 0,Y 501.781,Z 1041.443,A -85,B 0,C 180,E1 20299.208,E2 20299.208} C_VEL
LIN {X 0,Y 496.428,Z 1060.042,A -85,B 0,C 180,E1 20297.823,E2 20297.823} C_VEL
LIN {X 0,Y 491.098,Z 1077.508,A -85,B 0,C 180,E1 20296.353,E2 20296.353} C_VEL
LIN {X 0,Y 485.665,Z 1094.487,A -85,B 0,C 180,E1 20294.741,E2 20294.741} C_VEL
LIN {X 0,Y 479.684,Z 1112.577,A -85,B 0,C 180,E1 20292.797,E2 20292.797} C_VEL
LIN {X 0,Y 472.521,Z 1133.531,A -85,B 0,C 180,E1 20290.186,E2 20290.186} C_VEL
LIN {X 0,Y 467.295,Z 1148.548,A -85,B 0,C 180,E1 20288.033,E2 20288.033} C_VEL
LIN {X 0,Y 462.608,Z 1162.113,A -85,B 0,C 180,E1 20285.846,E2 20285.846} C_VEL
LIN {X 0,Y 458.191,Z 1175.065,A -85,B 0,C 180,E1 20283.503,E2 20283.503} C_VEL
LIN {X 0,Y 453.749,Z 1188.579,A -85,B 0,C 180,E1 20280.738,E2 20280.738} C_VEL
LIN {X 0,Y 449.434,Z 1202.497,A -85,B 0,C 180,E1 20277.413,E2 20277.413} C_VEL
LIN {X 0,Y 446.979,Z 1211.193,A -85,B 0,C 180,E1 20275.03,E2 20275.03} C_VEL
LIN {X 0,Y 445.175,Z 1214.364,A -85,B 0,C 180,E1 20274.149,E2 20274.149} C_VEL
LIN {X 0,Y 437.196,Z 1222.761,A -85,B 0,C 180,E1 20271.834,E2 20271.834} C_VEL
LIN {X 0,Y 435.884,Z 1225.064,A -85,B 0,C 180,E1 20271.03,E2 20271.03} C_VEL
LIN {X 0,Y 434.044,Z 1233.482,A -85,B 0,C 180,E1 20267.557,E2 20267.557} C_VEL
LIN {X 0,Y 433.064,Z 1239.001,A -85,B 0,C 180,E1 20264.843,E2 20264.843} C_VEL
LIN {X 0,Y 432.467,Z 1243.747,A -85,B 0,C 180,E1 20262.003,E2 20262.003} C_VEL
LIN {X 0,Y 432.109,Z 1247.312,A -85,B 0,C 180,E1 20259.315,E2 20259.315} C_VEL
LIN {X 0,Y 431.993,Z 1249.964,A -85,B 0,C 180,E1 20256.639,E2 20256.639} C_VEL
LIN {X 0,Y 431.932,Z 1251.727,A -85,B 0,C 180,E1 20253.976,E2 20253.976} C_VEL
LIN {X 0,Y 431.911,Z 1252.614,A -85,B 0,C 180,E1 20251.32,E2 20251.32} C_VEL
LIN {X 0,Y 431.903,Z 1252.627,A -85,B 0,C 180,E1 20248.667,E2 20248.667} C_VEL
LIN {X 0,Y 431.935,Z 1251.767,A -85,B 0,C 180,E1 20246.012,E2 20246.012} C_VEL
LIN {X 0,Y 431.989,Z 1250.029,A -85,B 0,C 180,E1 20243.349,E2 20243.349} C_VEL
LIN {X 0,Y 432.106,Z 1247.402,A -85,B 0,C 180,E1 20240.673,E2 20240.673} C_VEL
LIN {X 0,Y 432.454,Z 1243.842,A -85,B 0,C 180,E1 20237.97,E2 20237.97} C_VEL
LIN {X 0,Y 433.006,Z 1239.389,A -85,B 0,C 180,E1 20235.28,E2 20235.28} C_VEL
LIN {X 0,Y 433.969,Z 1233.872,A -85,B 0,C 180,E1 20232.532,E2 20232.532} C_VEL
LIN {X 0,Y 435.454,Z 1226.712,A -85,B 0,C 180,E1 20229.53,E2 20229.53} C_VEL
LIN {X 0,Y 438.103,Z 1216.274,A -85,B 0,C 180,E1 20225.882,E2 20225.882} C_VEL
LIN {X 0,Y 441.039,Z 1206.054,A -85,B 0,C 180,E1 20222.886,E2 20222.886} C_VEL
LIN {X 0,Y 444.383,Z 1195.485,A -85,B 0,C 180,E1 20220.176,E2 20220.176} C_VEL
LIN {X 0,Y 448.192,Z 1184.193,A -85,B 0,C 180,E1 20217.622,E2 20217.622} C_VEL
LIN {X 0,Y 453.38,Z 1169.457,A -85,B 0,C 180,E1 20214.687,E2 20214.687} C_VEL
LIN {X 0,Y 459.547,Z 1152.225,A -85,B 0,C 180,E1 20211.765,E2 20211.765} C_VEL
LIN {X 0,Y 464.798,Z 1137.68,A -85,B 0,C 180,E1 20209.6,E2 20209.6} C_VEL
LIN {X 0,Y 470.185,Z 1122.635,A -85,B 0,C 180,E1 20207.609,E2 20207.609} C_VEL
LIN {X 0,Y 476.141,Z 1105.715,A -85,B 0,C 180,E1 20205.625,E2 20205.625} C_VEL
LIN {X 0,Y 483.829,Z 1082.993,A -85,B 0,C 180,E1 20203.323,E2 20203.323} C_VEL
LIN {X 0,Y 489.89,Z 1063.917,A -85,B 0,C 180,E1 20201.662,E2 20201.662} C_VEL
LIN {X 0,Y 495.353,Z 1045.684,A -85,B 0,C 180,E1 20200.266,E2 20200.266} C_VEL
LIN {X 0,Y 500.684,Z 1026.611,A -85,B 0,C 180,E1 20198.982,E2 20198.982} C_VEL
LIN {X 0,Y 506.532,Z 1003.961,A -85,B 0,C 180,E1 20197.663,E2 20197.663} C_VEL
LIN {X 0,Y 512.436,Z 977.763,A -85,B 0,C 180,E1 20196.396,E2 20196.396} C_VEL
LIN {X 0,Y 516.538,Z 956.941,A -85,B 0,C 180,E1 20195.557,E2 20195.557} C_VEL
LIN {X 0,Y 520.076,Z 936.204,A -85,B 0,C 180,E1 20194.853,E2 20194.853} C_VEL
LIN {X 0,Y 523.196,Z 914.527,A -85,B 0,C 180,E1 20194.249,E2 20194.249} C_VEL
LIN {X 0,Y 526.057,Z 889.587,A -85,B 0,C 180,E1 20193.703,E2 20193.703} C_VEL
LIN {X 0,Y 528.582,Z 852.318,A -85,B 0,C 180,E1 20193.094,E2 20193.094} C_VEL
LIN {X 0,Y 541.075,Z 631.433,A -85,B 0,C 180,E1 20189.693,E2 20189.693} C_VEL
LIN {X 0,Y 545.439,Z 556.746,A -85,B 0,C 180,E1 20188.525,E2 20188.525} C_VEL
LIN {X 0,Y 535.147,Z 541.717,A -85,B 0,C 180,E1 20185.956,E2 20185.956} C_VEL
LIN {X 0,Y 526.754,Z 530.25,A -85,B 0,C 180,E1 20183.611,E2 20183.611} C_VEL
LIN {X 0,Y 520.142,Z 521.43,A -85,B 0,C 180,E1 20181.541,E2 20181.541} C_VEL
LIN {X 0,Y 516.295,Z 516.495,A -85,B 0,C 180,E1 20180.224,E2 20180.224} C_VEL
LIN {X 0,Y 512.274,Z 511.32,A -85,B 0,C 180,E1 20178.728,E2 20178.728} C_VEL
LIN {X 0,Y 508.303,Z 506.261,A -85,B 0,C 180,E1 20177.103,E2 20177.103} C_VEL
LIN {X 0,Y 504.688,Z 501.704,A -85,B 0,C 180,E1 20175.455,E2 20175.455} C_VEL
LIN {X 0,Y 500.308,Z 496.525,A -85,B 0,C 180,E1 20173.17,E2 20173.17} C_VEL
LIN {X 0,Y 499.387,Z 495.05,A -85,B 0,C 180,E1 20172.606,E2 20172.606} C_VEL
LIN {X 0,Y 496.044,Z 491.836,A -85,B 0,C 180,E1 20170.452,E2 20170.452} C_VEL
LIN {X 0,Y 494.406,Z 488.905,A -85,B 0,C 180,E1 20169.076,E2 20169.076} C_VEL
LIN {X 0,Y 490.79,Z 485.747,A -85,B 0,C 180,E1 20165.26,E2 20165.26} C_VEL
LIN {X 0,Y 489.73,Z 482.601,A -85,B 0,C 180,E1 20162.692,E2 20162.692} C_VEL
LIN {X 0,Y 489.788,Z 482.703,A -85,B 0,C 180,E1 20157.543,E2 20157.543} C_VEL
LIN {X 0,Y 491.682,Z 486.983,A -85,B 0,C 180,E1 20153.93,E2 20153.93} C_VEL
LIN {X 0,Y 494.755,Z 489.332,A -85,B 0,C 180,E1 20151.047,E2 20151.047} C_VEL
LIN {X 0,Y 497.086,Z 493.201,A -85,B 0,C 180,E1 20149.218,E2 20149.218} C_VEL
LIN {X 0,Y 499.772,Z 495.547,A -85,B 0,C 180,E1 20147.58,E2 20147.58} C_VEL
LIN {X 0,Y 502.988,Z 499.949,A -85,B 0,C 180,E1 20145.788,E2 20145.788} C_VEL
LIN {X 0,Y 504.583,Z 501.574,A -85,B 0,C 180,E1 20145.013,E2 20145.013} C_VEL
LIN {X 0,Y 508.18,Z 506.169,A -85,B 0,C 180,E1 20143.364,E2 20143.364} C_VEL
LIN {X 0,Y 512.444,Z 512.014,A -85,B 0,C 180,E1 20141.602,E2 20141.602} C_VEL
LIN {X 0,Y 516.799,Z 518.184,A -85,B 0,C 180,E1 20139.973,E2 20139.973} C_VEL
LIN {X 0,Y 522.152,Z 525.758,A -85,B 0,C 180,E1 20138.162,E2 20138.162} C_VEL
LIN {X 0,Y 531.334,Z 539.548,A -85,B 0,C 180,E1 20135.395,E2 20135.395} C_VEL
LIN {X 0,Y 540.286,Z 553.785,A -85,B 0,C 180,E1 20133.007,E2 20133.007} C_VEL
LIN {X 0,Y 545.543,Z 562.638,A -85,B 0,C 180,E1 20131.712,E2 20131.712} C_VEL
LIN {X 0,Y 533.329,Z 775.013,A -85,B 0,C 180,E1 20128.429,E2 20128.429} C_VEL
LIN {X 0,Y 526.339,Z 898.926,A -85,B 0,C 180,E1 20126.507,E2 20126.507} C_VEL
LIN {X 0,Y 523.61,Z 926.446,A -85,B 0,C 180,E1 20125.983,E2 20125.983} C_VEL
LIN {X 0,Y 519.765,Z 953.005,A -85,B 0,C 180,E1 20125.3,E2 20125.3} C_VEL
LIN {X 0,Y 516.059,Z 974.513,A -85,B 0,C 180,E1 20124.609,E2 20124.609} C_VEL
LIN {X 0,Y 512.009,Z 995.069,A -85,B 0,C 180,E1 20123.815,E2 20123.815} C_VEL
LIN {X 0,Y 507.37,Z 1016.017,A -85,B 0,C 180,E1 20122.864,E2 20122.864} C_VEL
LIN {X 0,Y 501.058,Z 1041.759,A -85,B 0,C 180,E1 20121.472,E2 20121.472} C_VEL
LIN {X 0,Y 495.007,Z 1063.677,A -85,B 0,C 180,E1 20120.063,E2 20120.063} C_VEL
LIN {X 0,Y 489.414,Z 1082.642,A -85,B 0,C 180,E1 20118.665,E2 20118.665} C_VEL
LIN {X 0,Y 483.829,Z 1100.606,A -85,B 0,C 180,E1 20117.163,E2 20117.163} C_VEL
LIN {X 0,Y 477.731,Z 1119.475,A -85,B 0,C 180,E1 20115.371,E2 20115.371} C_VEL
LIN {X 0,Y 469.989,Z 1142.542,A -85,B 0,C 180,E1 20112.827,E2 20112.827} C_VEL
LIN {X 0,Y 464.248,Z 1159.216,A -85,B 0,C 180,E1 20110.7,E2 20110.7} C_VEL
LIN {X 0,Y 459.041,Z 1174.282,A -85,B 0,C 180,E1 20108.538,E2 20108.538} C_VEL
LIN {X 0,Y 454.06,Z 1188.925,A -85,B 0,C 180,E1 20106.173,E2 20106.173} C_VEL
LIN {X 0,Y 448.376,Z 1206.031,A -85,B 0,C 180,E1 20103.019,E2 20103.019} C_VEL
LIN {X 0,Y 444.138,Z 1219.43,A -85,B 0,C 180,E1 20100.14,E2 20100.14} C_VEL
LIN {X 0,Y 440.826,Z 1230.598,A -85,B 0,C 180,E1 20097.421,E2 20097.421} C_VEL
LIN {X 0,Y 438.185,Z 1240.491,A -85,B 0,C 180,E1 20094.687,E2 20094.687} C_VEL
LIN {X 0,Y 435.684,Z 1251.256,A -85,B 0,C 180,E1 20091.266,E2 20091.266} C_VEL
LIN {X 0,Y 433.875,Z 1260.396,A -85,B 0,C 180,E1 20087.715,E2 20087.715} C_VEL
LIN {X 0,Y 432.918,Z 1266.533,A -85,B 0,C 180,E1 20084.86,E2 20084.86} C_VEL
LIN {X 0,Y 432.399,Z 1271.348,A -85,B 0,C 180,E1 20082.153,E2 20082.153} C_VEL
LIN {X 0,Y 432.063,Z 1275.175,A -85,B 0,C 180,E1 20079.463,E2 20079.463} C_VEL
LIN {X 0,Y 431.97,Z 1278.052,A -85,B 0,C 180,E1 20076.773,E2 20076.773} C_VEL
LIN {X 0,Y 431.926,Z 1279.96,A -85,B 0,C 180,E1 20074.121,E2 20074.121} C_VEL
LIN {X 0,Y 431.912,Z 1280.941,A -85,B 0,C 180,E1 20071.465,E2 20071.465} C_VEL
LIN {X 0,Y 431.891,Z 1281.013,A -85,B 0,C 180,E1 20068.945,E2 20068.945} C_VEL
LIN {X 0,Y 431.924,Z 1280.176,A -85,B 0,C 180,E1 20066.29,E2 20066.29} C_VEL
LIN {X 0,Y 431.963,Z 1278.403,A -85,B 0,C 180,E1 20063.627,E2 20063.627} C_VEL
LIN {X 0,Y 432.053,Z 1275.519,A -85,B 0,C 180,E1 20060.818,E2 20060.818} C_VEL
LIN {X 0,Y 432.356,Z 1271.793,A -85,B 0,C 180,E1 20058.129,E2 20058.129} C_VEL
LIN {X 0,Y 432.847,Z 1267.081,A -85,B 0,C 180,E1 20055.423,E2 20055.423} C_VEL
LIN {X 0,Y 433.721,Z 1261.359,A -85,B 0,C 180,E1 20052.706,E2 20052.706} C_VEL
LIN {X 0,Y 435.004,Z 1254.226,A -85,B 0,C 180,E1 20049.839,E2 20049.839} C_VEL
LIN {X 0,Y 437.06,Z 1245.068,A -85,B 0,C 180,E1 20046.693,E2 20046.693} C_VEL
LIN {X 0,Y 440.236,Z 1232.757,A -85,B 0,C 180,E1 20043.138,E2 20043.138} C_VEL
LIN {X 0,Y 443.402,Z 1221.827,A -85,B 0,C 180,E1 20040.414,E2 20040.414} C_VEL
LIN {X 0,Y 447.029,Z 1210.18,A -85,B 0,C 180,E1 20037.845,E2 20037.845} C_VEL
LIN {X 0,Y 451.256,Z 1197.16,A -85,B 0,C 180,E1 20035.292,E2 20035.292} C_VEL
LIN {X 0,Y 457.059,Z 1180.205,A -85,B 0,C 180,E1 20032.367,E2 20032.367} C_VEL
LIN {X 0,Y 463.166,Z 1162.326,A -85,B 0,C 180,E1 20029.727,E2 20029.727} C_VEL
LIN {X 0,Y 468.479,Z 1146.875,A -85,B 0,C 180,E1 20027.707,E2 20027.707} C_VEL
LIN {X 0,Y 473.944,Z 1130.785,A -85,B 0,C 180,E1 20025.833,E2 20025.833} C_VEL
LIN {X 0,Y 479.715,Z 1113.383,A -85,B 0,C 180,E1 20024.031,E2 20024.031} C_VEL
LIN {X 0,Y 486.952,Z 1090.867,A -85,B 0,C 180,E1 20021.997,E2 20021.997} C_VEL
LIN {X 0,Y 493.516,Z 1068.765,A -85,B 0,C 180,E1 20020.3,E2 20020.3} C_VEL
LIN {X 0,Y 498.751,Z 1049.999,A -85,B 0,C 180,E1 20019.039,E2 20019.039} C_VEL
LIN {X 0,Y 503.713,Z 1030.91,A -85,B 0,C 180,E1 20017.916,E2 20017.916} C_VEL
LIN {X 0,Y 508.356,Z 1011.549,A -85,B 0,C 180,E1 20016.926,E2 20016.926} C_VEL
LIN {X 0,Y 512.875,Z 990.694,A -85,B 0,C 180,E1 20016.008,E2 20016.008} C_VEL
LIN {X 0,Y 517.953,Z 964.015,A -85,B 0,C 180,E1 20015.035,E2 20015.035} C_VEL
LIN {X 0,Y 521.859,Z 938.612,A -85,B 0,C 180,E1 20014.314,E2 20014.314} C_VEL
LIN {X 0,Y 524.628,Z 916.527,A -85,B 0,C 180,E1 20013.821,E2 20013.821} C_VEL
LIN {X 0,Y 526.647,Z 893.914,A -85,B 0,C 180,E1 20013.414,E2 20013.414} C_VEL
LIN {X 0,Y 538.891,Z 675.325,A -85,B 0,C 180,E1 20010.038,E2 20010.038} C_VEL
LIN {X 0,Y 545.421,Z 562.342,A -85,B 0,C 180,E1 20008.277,E2 20008.277} C_VEL
LIN {X 0,Y 537.134,Z 548.901,A -85,B 0,C 180,E1 20006.213,E2 20006.213} C_VEL
LIN {X 0,Y 529.797,Z 537.405,A -85,B 0,C 180,E1 20004.206,E2 20004.206} C_VEL
LIN {X 0,Y 521.476,Z 524.815,A -85,B 0,C 180,E1 20001.66,E2 20001.66} C_VEL
LIN {X 0,Y 514.196,Z 514.531,A -85,B 0,C 180,E1 19999.127,E2 19999.127} C_VEL
LIN {X 0,Y 508.417,Z 506.459,A -85,B 0,C 180,E1 19996.804,E2 19996.804} C_VEL
LIN {X 0,Y 504.751,Z 501.994,A -85,B 0,C 180,E1 19995.158,E2 19995.158} C_VEL
LIN {X 0,Y 503.614,Z 500.57,A -85,B 0,C 180,E1 19994.605,E2 19994.605} C_VEL
LIN {X 0,Y 500.046,Z 496.229,A -85,B 0,C 180,E1 19992.706,E2 19992.706} C_VEL
LIN {X 0,Y 499.102,Z 494.948,A -85,B 0,C 180,E1 19992.143,E2 19992.143} C_VEL
LIN {X 0,Y 496.006,Z 491.927,A -85,B 0,C 180,E1 19990.16,E2 19990.16} C_VEL
LIN {X 0,Y 494.42,Z 488.938,A -85,B 0,C 180,E1 19988.841,E2 19988.841} C_VEL
LIN {X 0,Y 490.752,Z 485.904,A -85,B 0,C 180,E1 19985.143,E2 19985.143} C_VEL
LIN {X 0,Y 489.579,Z 482.596,A -85,B 0,C 180,E1 19982.575,E2 19982.575} C_VEL
LIN {X 0,Y 489.692,Z 482.817,A -85,B 0,C 180,E1 19976.605,E2 19976.605} C_VEL
LIN {X 0,Y 491.066,Z 486.277,A -85,B 0,C 180,E1 19973.922,E2 19973.922} C_VEL
LIN {X 0,Y 494.642,Z 489.323,A -85,B 0,C 180,E1 19970.459,E2 19970.459} C_VEL
LIN {X 0,Y 496.841,Z 492.988,A -85,B 0,C 180,E1 19968.743,E2 19968.743} C_VEL
LIN {X 0,Y 499.729,Z 495.605,A -85,B 0,C 180,E1 19966.985,E2 19966.985} C_VEL
LIN {X 0,Y 502.856,Z 499.906,A -85,B 0,C 180,E1 19965.255,E2 19965.255} C_VEL
LIN {X 0,Y 504.575,Z 501.68,A -85,B 0,C 180,E1 19964.424,E2 19964.424} C_VEL
LIN {X 0,Y 508.212,Z 506.215,A -85,B 0,C 180,E1 19962.776,E2 19962.776} C_VEL
LIN {X 0,Y 513.826,Z 513.331,A -85,B 0,C 180,E1 19960.534,E2 19960.534} C_VEL
LIN {X 0,Y 518.679,Z 519.629,A -85,B 0,C 180,E1 19958.81,E2 19958.81} C_VEL
LIN {X 0,Y 525.285,Z 528.219,A -85,B 0,C 180,E1 19956.705,E2 19956.705} C_VEL
LIN {X 0,Y 533.453,Z 539.516,A -85,B 0,C 180,E1 19954.373,E2 19954.373} C_VEL
LIN {X 0,Y 542.525,Z 552.521,A -85,B 0,C 180,E1 19952.057,E2 19952.057} C_VEL
LIN {X 0,Y 545.403,Z 557.054,A -85,B 0,C 180,E1 19951.363,E2 19951.363} C_VEL
LIN {X 0,Y 532.616,Z 778.055,A -85,B 0,C 180,E1 19947.954,E2 19947.954} C_VEL
LIN {X 0,Y 526.774,Z 880.199,A -85,B 0,C 180,E1 19946.366,E2 19946.366} C_VEL
LIN {X 0,Y 524.096,Z 907.512,A -85,B 0,C 180,E1 19945.831,E2 19945.831} C_VEL
LIN {X 0,Y 520.418,Z 933.71,A -85,B 0,C 180,E1 19945.13,E2 19945.13} C_VEL
LIN {X 0,Y 516.858,Z 954.896,A -85,B 0,C 180,E1 19944.424,E2 19944.424} C_VEL
LIN {X 0,Y 512.884,Z 975.343,A -85,B 0,C 180,E1 19943.613,E2 19943.613} C_VEL
LIN {X 0,Y 507.956,Z 997.745,A -85,B 0,C 180,E1 19942.564,E2 19942.564} C_VEL
LIN {X 0,Y 501.254,Z 1024.411,A -85,B 0,C 180,E1 19941.062,E2 19941.062} C_VEL
LIN {X 0,Y 495.772,Z 1044.128,A -85,B 0,C 180,E1 19939.75,E2 19939.75} C_VEL
LIN {X 0,Y 490.266,Z 1062.57,A -85,B 0,C 180,E1 19938.351,E2 19938.351} C_VEL
LIN {X 0,Y 484.836,Z 1079.718,A -85,B 0,C 180,E1 19936.88,E2 19936.88} C_VEL
LIN {X 0,Y 478.473,Z 1098.928,A -85,B 0,C 180,E1 19935.011,E2 19935.011} C_VEL
LIN {X 0,Y 471.078,Z 1120.148,A -85,B 0,C 180,E1 19932.606,E2 19932.606} C_VEL
LIN {X 0,Y 465.362,Z 1136.087,A -85,B 0,C 180,E1 19930.528,E2 19930.528} C_VEL
LIN {X 0,Y 460.158,Z 1150.488,A -85,B 0,C 180,E1 19928.413,E2 19928.413} C_VEL
LIN {X 0,Y 454.977,Z 1164.897,A -85,B 0,C 180,E1 19926.026,E2 19926.026} C_VEL
LIN {X 0,Y 449.181,Z 1181.384,A -85,B 0,C 180,E1 19922.889,E2 19922.889} C_VEL
LIN {X 0,Y 444.671,Z 1194.634,A -85,B 0,C 180,E1 19919.938,E2 19919.938} C_VEL
LIN {X 0,Y 441.42,Z 1204.786,A -85,B 0,C 180,E1 19917.368,E2 19917.368} C_VEL
LIN {X 0,Y 438.656,Z 1214.242,A -85,B 0,C 180,E1 19914.646,E2 19914.646} C_VEL
LIN {X 0,Y 436.023,Z 1224.499,A -85,B 0,C 180,E1 19911.235,E2 19911.235} C_VEL
LIN {X 0,Y 435.884,Z 1225.064,A -85,B 0,C 180,E1 19911.03,E2 19911.03} C_VEL
LIN {X 0,Y 434.279,Z 1227.655,A -85,B 0,C 180,E1 19910.086,E2 19910.086} C_VEL
LIN {X 0,Y 426.678,Z 1234.478,A -85,B 0,C 180,E1 19907.52,E2 19907.52} C_VEL
LIN {X 0,Y 425.748,Z 1236.196,A -85,B 0,C 180,E1 19906.742,E2 19906.742} C_VEL
LIN {X 0,Y 424.636,Z 1243.077,A -85,B 0,C 180,E1 19902.877,E2 19902.877} C_VEL
LIN {X 0,Y 424.174,Z 1247.114,A -85,B 0,C 180,E1 19899.902,E2 19899.902} C_VEL
LIN {X 0,Y 424.01,Z 1250.009,A -85,B 0,C 180,E1 19897.037,E2 19897.037} C_VEL
LIN {X 0,Y 423.941,Z 1251.859,A -85,B 0,C 180,E1 19894.322,E2 19894.322} C_VEL
LIN {X 0,Y 423.923,Z 1252.833,A -85,B 0,C 180,E1 19891.616,E2 19891.616} C_VEL
LIN {X 0,Y 423.895,Z 1252.934,A -85,B 0,C 180,E1 19888.913,E2 19888.913} C_VEL
LIN {X 0,Y 423.939,Z 1252.161,A -85,B 0,C 180,E1 19886.207,E2 19886.207} C_VEL
LIN {X 0,Y 423.998,Z 1250.402,A -85,B 0,C 180,E1 19883.359,E2 19883.359} C_VEL
LIN {X 0,Y 424.12,Z 1247.822,A -85,B 0,C 180,E1 19880.632,E2 19880.632} C_VEL
LIN {X 0,Y 424.484,Z 1244.329,A -85,B 0,C 180,E1 19877.893,E2 19877.893} C_VEL
LIN {X 0,Y 425.067,Z 1239.902,A -85,B 0,C 180,E1 19875.138,E2 19875.138} C_VEL
LIN {X 0,Y 426.089,Z 1234.388,A -85,B 0,C 180,E1 19872.317,E2 19872.317} C_VEL
LIN {X 0,Y 427.53,Z 1227.76,A -85,B 0,C 180,E1 19869.458,E2 19869.458} C_VEL
LIN {X 0,Y 429.712,Z 1219.457,A -85,B 0,C 180,E1 19866.403,E2 19866.403} C_VEL
LIN {X 0,Y 433.33,Z 1207.332,A -85,B 0,C 180,E1 19862.661,E2 19862.661} C_VEL
LIN {X 0,Y 436.976,Z 1196.317,A -85,B 0,C 180,E1 19859.77,E2 19859.77} C_VEL
LIN {X 0,Y 440.937,Z 1185.088,A -85,B 0,C 180,E1 19857.177,E2 19857.177} C_VEL
LIN {X 0,Y 445.672,Z 1172.105,A -85,B 0,C 180,E1 19854.53,E2 19854.53} C_VEL
LIN {X 0,Y 452.296,Z 1154.503,A -85,B 0,C 180,E1 19851.429,E2 19851.429} C_VEL
LIN {X 0,Y 458.243,Z 1138.634,A -85,B 0,C 180,E1 19849.024,E2 19849.024} C_VEL
LIN {X 0,Y 463.91,Z 1123.403,A -85,B 0,C 180,E1 19846.982,E2 19846.982} C_VEL
LIN {X 0,Y 469.865,Z 1107.078,A -85,B 0,C 180,E1 19845.044,E2 19845.044} C_VEL
LIN {X 0,Y 477.363,Z 1085.9,A -85,B 0,C 180,E1 19842.848,E2 19842.848} C_VEL
LIN {X 0,Y 484.248,Z 1064.909,A -85,B 0,C 180,E1 19840.997,E2 19840.997} C_VEL
LIN {X 0,Y 489.871,Z 1046.75,A -85,B 0,C 180,E1 19839.595,E2 19839.595} C_VEL
LIN {X 0,Y 495.262,Z 1028.078,A -85,B 0,C 180,E1 19838.326,E2 19838.326} C_VEL
LIN {X 0,Y 500.575,Z 1008.209,A -85,B 0,C 180,E1 19837.152,E2 19837.152} C_VEL
LIN {X 0,Y 506.369,Z 984.307,A -85,B 0,C 180,E1 19835.939,E2 19835.939} C_VEL
LIN {X 0,Y 511.622,Z 958.667,A -85,B 0,C 180,E1 19834.877,E2 19834.877} C_VEL
LIN {X 0,Y 515.385,Z 937.319,A -85,B 0,C 180,E1 19834.146,E2 19834.146} C_VEL
LIN {X 0,Y 518.563,Z 915.944,A -85,B 0,C 180,E1 19833.546,E2 19833.546} C_VEL
LIN {X 0,Y 521.231,Z 893.621,A -85,B 0,C 180,E1 19833.047,E2 19833.047} C_VEL
LIN {X 0,Y 523.744,Z 861.586,A -85,B 0,C 180,E1 19832.5,E2 19832.5} C_VEL
LIN {X 0,Y 536.638,Z 640.166,A -85,B 0,C 180,E1 19829.082,E2 19829.082} C_VEL
LIN {X 0,Y 541.406,Z 561.492,A -85,B 0,C 180,E1 19827.856,E2 19827.856} C_VEL
LIN {X 0,Y 532.008,Z 547.727,A -85,B 0,C 180,E1 19825.433,E2 19825.433} C_VEL
LIN {X 0,Y 522.904,Z 534.948,A -85,B 0,C 180,E1 19822.782,E2 19822.782} C_VEL
LIN {X 0,Y 515.177,Z 524.716,A -85,B 0,C 180,E1 19820.211,E2 19820.211} C_VEL
LIN {X 0,Y 510.468,Z 518.715,A -85,B 0,C 180,E1 19818.442,E2 19818.442} C_VEL
LIN {X 0,Y 506.564,Z 513.707,A -85,B 0,C 180,E1 19816.808,E2 19816.808} C_VEL
LIN {X 0,Y 502.471,Z 508.436,A -85,B 0,C 180,E1 19814.875,E2 19814.875} C_VEL
LIN {X 0,Y 499.034,Z 504.38,A -85,B 0,C 180,E1 19813.027,E2 19813.027} C_VEL
LIN {X 0,Y 498.031,Z 502.809,A -85,B 0,C 180,E1 19812.405,E2 19812.405} C_VEL
LIN {X 0,Y 494.762,Z 499.528,A -85,B 0,C 180,E1 19810.244,E2 19810.244} C_VEL
LIN {X 0,Y 493.296,Z 496.797,A -85,B 0,C 180,E1 19808.979,E2 19808.979} C_VEL
LIN {X 0,Y 489.671,Z 493.496,A -85,B 0,C 180,E1 19805.037,E2 19805.037} C_VEL
LIN {X 0,Y 488.715,Z 490.535,A -85,B 0,C 180,E1 19802.58,E2 19802.58} C_VEL
LIN {X 0,Y 488.799,Z 490.765,A -85,B 0,C 180,E1 19797.538,E2 19797.538} C_VEL
LIN {X 0,Y 490.707,Z 494.966,A -85,B 0,C 180,E1 19793.918,E2 19793.918} C_VEL
LIN {X 0,Y 493.566,Z 497.175,A -85,B 0,C 180,E1 19791.202,E2 19791.202} C_VEL
LIN {X 0,Y 495.944,Z 501.091,A -85,B 0,C 180,E1 19789.311,E2 19789.311} C_VEL
LIN {X 0,Y 498.5,Z 503.43,A -85,B 0,C 180,E1 19787.724,E2 19787.724} C_VEL
LIN {X 0,Y 501.798,Z 507.855,A -85,B 0,C 180,E1 19785.872,E2 19785.872} C_VEL
LIN {X 0,Y 503.253,Z 509.491,A -85,B 0,C 180,E1 19785.149,E2 19785.149} C_VEL
LIN {X 0,Y 508.473,Z 516.219,A -85,B 0,C 180,E1 19782.785,E2 19782.785} C_VEL
LIN {X 0,Y 514.483,Z 524.901,A -85,B 0,C 180,E1 19780.412,E2 19780.412} C_VEL
LIN {X 0,Y 520.111,Z 533.022,A -85,B 0,C 180,E1 19778.458,E2 19778.458} C_VEL
LIN {X 0,Y 529.073,Z 546.716,A -85,B 0,C 180,E1 19775.699,E2 19775.699} C_VEL
LIN {X 0,Y 537.906,Z 560.977,A -85,B 0,C 180,E1 19773.296,E2 19773.296} C_VEL
LIN {X 0,Y 541.473,Z 567.193,A -85,B 0,C 180,E1 19772.388,E2 19772.388} C_VEL
LIN {X 0,Y 528.847,Z 780.158,A -85,B 0,C 180,E1 19769.089,E2 19769.089} C_VEL
LIN {X 0,Y 521.931,Z 898.788,A -85,B 0,C 180,E1 19767.242,E2 19767.242} C_VEL
LIN {X 0,Y 519.125,Z 926.334,A -85,B 0,C 180,E1 19766.717,E2 19766.717} C_VEL
LIN {X 0,Y 515.18,Z 952.878,A -85,B 0,C 180,E1 19766.036,E2 19766.036} C_VEL
LIN {X 0,Y 511.418,Z 974.182,A -85,B 0,C 180,E1 19765.352,E2 19765.352} C_VEL
LIN {X 0,Y 507.263,Z 994.696,A -85,B 0,C 180,E1 19764.563,E2 19764.563} C_VEL
LIN {X 0,Y 502.501,Z 1015.641,A -85,B 0,C 180,E1 19763.613,E2 19763.613} C_VEL
LIN {X 0,Y 496.231,Z 1040.586,A -85,B 0,C 180,E1 19762.272,E2 19762.272} C_VEL
LIN {X 0,Y 489.7,Z 1063.52,A -85,B 0,C 180,E1 19760.798,E2 19760.798} C_VEL
LIN {X 0,Y 483.732,Z 1083.115,A -85,B 0,C 180,E1 19759.345,E2 19759.345} C_VEL
LIN {X 0,Y 477.847,Z 1101.416,A -85,B 0,C 180,E1 19757.799,E2 19757.799} C_VEL
LIN {X 0,Y 470.677,Z 1122.897,A -85,B 0,C 180,E1 19755.722,E2 19755.722} C_VEL
LIN {X 0,Y 463.476,Z 1143.296,A -85,B 0,C 180,E1 19753.407,E2 19753.407} C_VEL
LIN {X 0,Y 457.879,Z 1158.936,A -85,B 0,C 180,E1 19751.39,E2 19751.39} C_VEL
LIN {X 0,Y 452.459,Z 1174.007,A -85,B 0,C 180,E1 19749.205,E2 19749.205} C_VEL
LIN {X 0,Y 447.258,Z 1188.65,A -85,B 0,C 180,E1 19746.813,E2 19746.813} C_VEL
LIN {X 0,Y 441.235,Z 1205.962,A -85,B 0,C 180,E1 19743.573,E2 19743.573} C_VEL
LIN {X 0,Y 436.692,Z 1219.652,A -85,B 0,C 180,E1 19740.579,E2 19740.579} C_VEL
LIN {X 0,Y 433.346,Z 1230.431,A -85,B 0,C 180,E1 19737.905,E2 19737.905} C_VEL
LIN {X 0,Y 430.508,Z 1240.506,A -85,B 0,C 180,E1 19735.067,E2 19735.067} C_VEL
LIN {X 0,Y 427.847,Z 1251.382,A -85,B 0,C 180,E1 19731.531,E2 19731.531} C_VEL
LIN {X 0,Y 426.002,Z 1260.125,A -85,B 0,C 180,E1 19728.054,E2 19728.054} C_VEL
LIN {X 0,Y 424.997,Z 1266.264,A -85,B 0,C 180,E1 19725.144,E2 19725.144} C_VEL
LIN {X 0,Y 424.431,Z 1271.08,A -85,B 0,C 180,E1 19722.385,E2 19722.385} C_VEL
LIN {X 0,Y 424.088,Z 1274.774,A -85,B 0,C 180,E1 19719.755,E2 19719.755} C_VEL
LIN {X 0,Y 423.98,Z 1277.659,A -85,B 0,C 180,E1 19717.05,E2 19717.05} C_VEL
LIN {X 0,Y 423.93,Z 1279.626,A -85,B 0,C 180,E1 19714.334,E2 19714.334} C_VEL
LIN {X 0,Y 423.92,Z 1280.655,A -85,B 0,C 180,E1 19711.628,E2 19711.628} C_VEL
LIN {X 0,Y 423.896,Z 1280.75,A -85,B 0,C 180,E1 19708.925,E2 19708.925} C_VEL
LIN {X 0,Y 423.927,Z 1279.913,A -85,B 0,C 180,E1 19706.22,E2 19706.22} C_VEL
LIN {X 0,Y 423.967,Z 1278.139,A -85,B 0,C 180,E1 19703.507,E2 19703.507} C_VEL
LIN {X 0,Y 424.054,Z 1275.418,A -85,B 0,C 180,E1 19700.78,E2 19700.78} C_VEL
LIN {X 0,Y 424.368,Z 1271.738,A -85,B 0,C 180,E1 19698.04,E2 19698.04} C_VEL
LIN {X 0,Y 424.878,Z 1267.074,A -85,B 0,C 180,E1 19695.283,E2 19695.283} C_VEL
LIN {X 0,Y 425.789,Z 1261.4,A -85,B 0,C 180,E1 19692.515,E2 19692.515} C_VEL
LIN {X 0,Y 427.056,Z 1254.678,A -85,B 0,C 180,E1 19689.733,E2 19689.733} C_VEL
LIN {X 0,Y 428.868,Z 1246.869,A -85,B 0,C 180,E1 19686.949,E2 19686.949} C_VEL
LIN {X 0,Y 431.492,Z 1236.975,A -85,B 0,C 180,E1 19683.886,E2 19683.886} C_VEL
LIN {X 0,Y 435.726,Z 1222.72,A -85,B 0,C 180,E1 19680.143,E2 19680.143} C_VEL
LIN {X 0,Y 439.681,Z 1210.549,A -85,B 0,C 180,E1 19677.396,E2 19677.396} C_VEL
LIN {X 0,Y 444.063,Z 1197.618,A -85,B 0,C 180,E1 19674.81,E2 19674.81} C_VEL
LIN {X 0,Y 449.456,Z 1182.433,A -85,B 0,C 180,E1 19672.13,E2 19672.13} C_VEL
LIN {X 0,Y 456.432,Z 1162.986,A -85,B 0,C 180,E1 19669.173,E2 19669.173} C_VEL
LIN {X 0,Y 462.161,Z 1146.954,A -85,B 0,C 180,E1 19667.05,E2 19667.05} C_VEL
LIN {X 0,Y 467.834,Z 1130.872,A -85,B 0,C 180,E1 19665.157,E2 19665.157} C_VEL
LIN {X 0,Y 473.733,Z 1113.721,A -85,B 0,C 180,E1 19663.366,E2 19663.366} C_VEL
LIN {X 0,Y 480.972,Z 1092.02,A -85,B 0,C 180,E1 19661.38,E2 19661.38} C_VEL
LIN {X 0,Y 487.962,Z 1069.307,A -85,B 0,C 180,E1 19659.617,E2 19659.617} C_VEL
LIN {X 0,Y 493.529,Z 1049.995,A -85,B 0,C 180,E1 19658.313,E2 19658.313} C_VEL
LIN {X 0,Y 498.708,Z 1030.635,A -85,B 0,C 180,E1 19657.171,E2 19657.171} C_VEL
LIN {X 0,Y 503.485,Z 1011.275,A -85,B 0,C 180,E1 19656.182,E2 19656.182} C_VEL
LIN {X 0,Y 508.285,Z 989.709,A -85,B 0,C 180,E1 19655.236,E2 19655.236} C_VEL
LIN {X 0,Y 513.628,Z 961.981,A -85,B 0,C 180,E1 19654.241,E2 19654.241} C_VEL
LIN {X 0,Y 517.424,Z 937.789,A -85,B 0,C 180,E1 19653.561,E2 19653.561} C_VEL
LIN {X 0,Y 520.225,Z 915.923,A -85,B 0,C 180,E1 19653.078,E2 19653.078} C_VEL
LIN {X 0,Y 522.301,Z 892.995,A -85,B 0,C 180,E1 19652.665,E2 19652.665} C_VEL
LIN {X 0,Y 534.971,Z 673.859,A -85,B 0,C 180,E1 19649.273,E2 19649.273} C_VEL
LIN {X 0,Y 541.316,Z 566.827,A -85,B 0,C 180,E1 19647.592,E2 19647.592} C_VEL
LIN {X 0,Y 532.019,Z 551.499,A -85,B 0,C 180,E1 19645.165,E2 19645.165} C_VEL
LIN {X 0,Y 523.97,Z 539.05,A -85,B 0,C 180,E1 19642.822,E2 19642.822} C_VEL
LIN {X 0,Y 516.436,Z 527.675,A -85,B 0,C 180,E1 19640.337,E2 19640.337} C_VEL
LIN {X 0,Y 509.103,Z 517.206,A -85,B 0,C 180,E1 19637.546,E2 19637.546} C_VEL
LIN {X 0,Y 506.154,Z 513.41,A -85,B 0,C 180,E1 19636.291,E2 19636.291} C_VEL
LIN {X 0,Y 502.189,Z 508.271,A -85,B 0,C 180,E1 19634.411,E2 19634.411} C_VEL
LIN {X 0,Y 498.587,Z 503.771,A -85,B 0,C 180,E1 19632.45,E2 19632.45} C_VEL
LIN {X 0,Y 497.745,Z 502.702,A -85,B 0,C 180,E1 19631.941,E2 19631.941} C_VEL
LIN {X 0,Y 494.644,Z 499.499,A -85,B 0,C 180,E1 19629.894,E2 19629.894} C_VEL
LIN {X 0,Y 493.157,Z 496.77,A -85,B 0,C 180,E1 19628.629,E2 19628.629} C_VEL
LIN {X 0,Y 489.621,Z 493.646,A -85,B 0,C 180,E1 19624.92,E2 19624.92} C_VEL
LIN {X 0,Y 488.558,Z 490.531,A -85,B 0,C 180,E1 19622.463,E2 19622.463} C_VEL
LIN {X 0,Y 488.671,Z 490.704,A -85,B 0,C 180,E1 19616.716,E2 19616.716} C_VEL
LIN {X 0,Y 490.004,Z 494.157,A -85,B 0,C 180,E1 19614.026,E2 19614.026} C_VEL
LIN {X 0,Y 493.451,Z 497.173,A -85,B 0,C 180,E1 19610.612,E2 19610.612} C_VEL
LIN {X 0,Y 495.701,Z 500.881,A -85,B 0,C 180,E1 19608.834,E2 19608.834} C_VEL
LIN {X 0,Y 498.358,Z 503.307,A -85,B 0,C 180,E1 19607.191,E2 19607.191} C_VEL
LIN {X 0,Y 501.556,Z 507.709,A -85,B 0,C 180,E1 19605.393,E2 19605.393} C_VEL
LIN {X 0,Y 503.135,Z 509.413,A -85,B 0,C 180,E1 19604.615,E2 19604.615} C_VEL
LIN {X 0,Y 506.86,Z 514.024,A -85,B 0,C 180,E1 19602.906,E2 19602.906} C_VEL
LIN {X 0,Y 512.27,Z 521.109,A -85,B 0,C 180,E1 19600.71,E2 19600.71} C_VEL
LIN {X 0,Y 516.846,Z 527.099,A -85,B 0,C 180,E1 19599.058,E2 19599.058} C_VEL
LIN {X 0,Y 523.199,Z 535.491,A -85,B 0,C 180,E1 19596.994,E2 19596.994} C_VEL
LIN {X 0,Y 531.261,Z 546.796,A -85,B 0,C 180,E1 19594.648,E2 19594.648} C_VEL
LIN {X 0,Y 540.028,Z 559.553,A -85,B 0,C 180,E1 19592.366,E2 19592.366} C_VEL
LIN {X 0,Y 541.339,Z 561.758,A -85,B 0,C 180,E1 19592.038,E2 19592.038} C_VEL
LIN {X 0,Y 528.141,Z 783.037,A -85,B 0,C 180,E1 19588.617,E2 19588.617} C_VEL
LIN {X 0,Y 522.379,Z 880.518,A -85,B 0,C 180,E1 19587.097,E2 19587.097} C_VEL
LIN {X 0,Y 519.619,Z 907.921,A -85,B 0,C 180,E1 19586.559,E2 19586.559} C_VEL
LIN {X 0,Y 515.868,Z 933.985,A -85,B 0,C 180,E1 19585.861,E2 19585.861} C_VEL
LIN {X 0,Y 512.215,Z 955.171,A -85,B 0,C 180,E1 19585.157,E2 19585.157} C_VEL
LIN {X 0,Y 508.136,Z 975.617,A -85,B 0,C 180,E1 19584.345,E2 19584.345} C_VEL
LIN {X 0,Y 503.098,Z 997.907,A -85,B 0,C 180,E1 19583.303,E2 19583.303} C_VEL
LIN {X 0,Y 496.182,Z 1024.684,A -85,B 0,C 180,E1 19581.792,E2 19581.792} C_VEL
LIN {X 0,Y 490.537,Z 1044.401,A -85,B 0,C 180,E1 19580.478,E2 19580.478} C_VEL
LIN {X 0,Y 485.111,Z 1062.045,A -85,B 0,C 180,E1 19579.139,E2 19579.139} C_VEL
LIN {X 0,Y 479.432,Z 1079.42,A -85,B 0,C 180,E1 19577.651,E2 19577.651} C_VEL
LIN {X 0,Y 473.068,Z 1098.002,A -85,B 0,C 180,E1 19575.843,E2 19575.843} C_VEL
LIN {X 0,Y 465.204,Z 1119.924,A -85,B 0,C 180,E1 19573.36,E2 19573.36} C_VEL
LIN {X 0,Y 459.079,Z 1136.364,A -85,B 0,C 180,E1 19571.202,E2 19571.202} C_VEL
LIN {X 0,Y 453.662,Z 1150.764,A -85,B 0,C 180,E1 19569.066,E2 19569.066} C_VEL
LIN {X 0,Y 448.353,Z 1164.937,A -85,B 0,C 180,E1 19566.694,E2 19566.694} C_VEL
LIN {X 0,Y 442.426,Z 1181.038,A -85,B 0,C 180,E1 19563.612,E2 19563.612} C_VEL
LIN {X 0,Y 437.492,Z 1194.843,A -85,B 0,C 180,E1 19560.499,E2 19560.499} C_VEL
LIN {X 0,Y 433.916,Z 1205.457,A -85,B 0,C 180,E1 19557.764,E2 19557.764} C_VEL
LIN {X 0,Y 430.994,Z 1214.964,A -85,B 0,C 180,E1 19554.967,E2 19554.967} C_VEL
LIN {X 0,Y 428.141,Z 1225.508,A -85,B 0,C 180,E1 19551.358,E2 19551.358} C_VEL
LIN {X 0,Y 426.212,Z 1233.753,A -85,B 0,C 180,E1 19547.891,E2 19547.891} C_VEL
LIN {X 0,Y 425.748,Z 1236.196,A -85,B 0,C 180,E1 19546.742,E2 19546.742} C_VEL
LIN {X 0,Y 424.415,Z 1238.298,A -85,B 0,C 180,E1 19545.751,E2 19545.751} C_VEL
LIN {X 0,Y 417.322,Z 1243.455,A -85,B 0,C 180,E1 19543.026,E2 19543.026} C_VEL
LIN {X 0,Y 416.536,Z 1244.656,A -85,B 0,C 180,E1 19542.208,E2 19542.208} C_VEL
LIN {X 0,Y 416.133,Z 1248.308,A -85,B 0,C 180,E1 19539.257,E2 19539.257} C_VEL
LIN {X 0,Y 415.991,Z 1251.153,A -85,B 0,C 180,E1 19536.064,E2 19536.064} C_VEL
LIN {X 0,Y 415.932,Z 1252.966,A -85,B 0,C 180,E1 19532.474,E2 19532.474} C_VEL
LIN {X 0,Y 415.89,Z 1253.241,A -85,B 0,C 180,E1 19529.167,E2 19529.167} C_VEL
LIN {X 0,Y 415.943,Z 1252.49,A -85,B 0,C 180,E1 19526.272,E2 19526.272} C_VEL
LIN {X 0,Y 416.006,Z 1250.776,A -85,B 0,C 180,E1 19523.369,E2 19523.369} C_VEL
LIN {X 0,Y 416.143,Z 1248.086,A -85,B 0,C 180,E1 19520.451,E2 19520.451} C_VEL
LIN {X 0,Y 416.544,Z 1244.594,A -85,B 0,C 180,E1 19517.659,E2 19517.659} C_VEL
LIN {X 0,Y 417.175,Z 1240.169,A -85,B 0,C 180,E1 19514.85,E2 19514.85} C_VEL
LIN {X 0,Y 418.239,Z 1234.774,A -85,B 0,C 180,E1 19512.032,E2 19512.032} C_VEL
LIN {X 0,Y 419.719,Z 1228.373,A -85,B 0,C 180,E1 19509.204,E2 19509.204} C_VEL
LIN {X 0,Y 421.768,Z 1220.912,A -85,B 0,C 180,E1 19506.376,E2 19506.376} C_VEL
LIN {X 0,Y 425.175,Z 1210.093,A -85,B 0,C 180,E1 19502.851,E2 19502.851} C_VEL
LIN {X 0,Y 429.391,Z 1197.712,A -85,B 0,C 180,E1 19499.488,E2 19499.488} C_VEL
LIN {X 0,Y 433.707,Z 1185.982,A -85,B 0,C 180,E1 19496.717,E2 19496.717} C_VEL
LIN {X 0,Y 438.458,Z 1173.487,A -85,B 0,C 180,E1 19494.116,E2 19494.116} C_VEL
LIN {X 0,Y 444.877,Z 1157.254,A -85,B 0,C 180,E1 19491.161,E2 19491.161} C_VEL
LIN {X 0,Y 451.826,Z 1139.358,A -85,B 0,C 180,E1 19488.397,E2 19488.397} C_VEL
LIN {X 0,Y 457.693,Z 1124.171,A -85,B 0,C 180,E1 19486.338,E2 19486.338} C_VEL
LIN {X 0,Y 463.637,Z 1108.441,A -85,B 0,C 180,E1 19484.447,E2 19484.447} C_VEL
LIN {X 0,Y 470.156,Z 1090.615,A -85,B 0,C 180,E1 19482.555,E2 19482.555} C_VEL
LIN {X 0,Y 478.203,Z 1067.354,A -85,B 0,C 180,E1 19480.434,E2 19480.434} C_VEL
LIN {X 0,Y 484.458,Z 1047.817,A -85,B 0,C 180,E1 19478.908,E2 19478.908} C_VEL
LIN {X 0,Y 489.971,Z 1029.321,A -85,B 0,C 180,E1 19477.642,E2 19477.642} C_VEL
LIN {X 0,Y 495.448,Z 1009.466,A -85,B 0,C 180,E1 19476.459,E2 19476.459} C_VEL
LIN {X 0,Y 500.799,Z 988.046,A -85,B 0,C 180,E1 19475.358,E2 19475.358} C_VEL
LIN {X 0,Y 506.779,Z 960.393,A -85,B 0,C 180,E1 19474.184,E2 19474.184} C_VEL
LIN {X 0,Y 510.827,Z 938.111,A -85,B 0,C 180,E1 19473.417,E2 19473.417} C_VEL
LIN {X 0,Y 514.1,Z 916.712,A -85,B 0,C 180,E1 19472.814,E2 19472.814} C_VEL
LIN {X 0,Y 516.796,Z 894.838,A -85,B 0,C 180,E1 19472.322,E2 19472.322} C_VEL
LIN {X 0,Y 519.228,Z 866.263,A -85,B 0,C 180,E1 19471.824,E2 19471.824} C_VEL
LIN {X 0,Y 532.539,Z 644.385,A -85,B 0,C 180,E1 19468.39,E2 19468.39} C_VEL
LIN {X 0,Y 537.37,Z 566.183,A -85,B 0,C 180,E1 19467.159,E2 19467.159} C_VEL
LIN {X 0,Y 527.406,Z 551.464,A -85,B 0,C 180,E1 19464.472,E2 19464.472} C_VEL
LIN {X 0,Y 519.124,Z 540.011,A -85,B 0,C 180,E1 19461.942,E2 19461.942} C_VEL
LIN {X 0,Y 513.158,Z 531.926,A -85,B 0,C 180,E1 19459.878,E2 19459.878} C_VEL
LIN {X 0,Y 508.539,Z 525.952,A -85,B 0,C 180,E1 19458.099,E2 19458.099} C_VEL
LIN {X 0,Y 504.965,Z 521.271,A -85,B 0,C 180,E1 19456.567,E2 19456.567} C_VEL
LIN {X 0,Y 500.827,Z 515.946,A -85,B 0,C 180,E1 19454.57,E2 19454.57} C_VEL
LIN {X 0,Y 497.492,Z 511.77,A -85,B 0,C 180,E1 19452.714,E2 19452.714} C_VEL
LIN {X 0,Y 496.682,Z 510.564,A -85,B 0,C 180,E1 19452.203,E2 19452.203} C_VEL
LIN {X 0,Y 493.376,Z 507.039,A -85,B 0,C 180,E1 19449.945,E2 19449.945} C_VEL
LIN {X 0,Y 492.045,Z 504.623,A -85,B 0,C 180,E1 19448.767,E2 19448.767} C_VEL
LIN {X 0,Y 488.558,Z 501.245,A -85,B 0,C 180,E1 19444.813,E2 19444.813} C_VEL
LIN {X 0,Y 487.701,Z 498.469,A -85,B 0,C 180,E1 19442.468,E2 19442.468} C_VEL
LIN {X 0,Y 487.786,Z 498.649,A -85,B 0,C 180,E1 19437.65,E2 19437.65} C_VEL
LIN {X 0,Y 489.636,Z 502.846,A -85,B 0,C 180,E1 19434.022,E2 19434.022} C_VEL
LIN {X 0,Y 492.382,Z 505.013,A -85,B 0,C 180,E1 19431.357,E2 19431.357} C_VEL
LIN {X 0,Y 494.804,Z 508.98,A -85,B 0,C 180,E1 19429.403,E2 19429.403} C_VEL
LIN {X 0,Y 497.233,Z 511.302,A -85,B 0,C 180,E1 19427.869,E2 19427.869} C_VEL
LIN {X 0,Y 500.61,Z 515.758,A -85,B 0,C 180,E1 19425.955,E2 19425.955} C_VEL
LIN {X 0,Y 502.034,Z 517.571,A -85,B 0,C 180,E1 19425.23,E2 19425.23} C_VEL
LIN {X 0,Y 506.844,Z 523.765,A -85,B 0,C 180,E1 19423.024,E2 19423.024} C_VEL
LIN {X 0,Y 512.764,Z 532.48,A -85,B 0,C 180,E1 19420.64,E2 19420.64} C_VEL
LIN {X 0,Y 518.239,Z 540.532,A -85,B 0,C 180,E1 19418.702,E2 19418.702} C_VEL
LIN {X 0,Y 526.827,Z 553.88,A -85,B 0,C 180,E1 19416.006,E2 19416.006} C_VEL
LIN {X 0,Y 535.826,Z 568.622,A -85,B 0,C 180,E1 19413.513,E2 19413.513} C_VEL
LIN {X 0,Y 537.479,Z 571.77,A -85,B 0,C 180,E1 19413.074,E2 19413.074} C_VEL
LIN {X 0,Y 524.446,Z 785.096,A -85,B 0,C 180,E1 19409.763,E2 19409.763} C_VEL
LIN {X 0,Y 517.619,Z 898.543,A -85,B 0,C 180,E1 19407.991,E2 19407.991} C_VEL
LIN {X 0,Y 514.746,Z 926.082,A -85,B 0,C 180,E1 19407.467,E2 19407.467} C_VEL
LIN {X 0,Y 510.705,Z 952.622,A -85,B 0,C 180,E1 19406.789,E2 19406.789} C_VEL
LIN {X 0,Y 506.837,Z 973.998,A -85,B 0,C 180,E1 19406.104,E2 19406.104} C_VEL
LIN {X 0,Y 502.579,Z 994.452,A -85,B 0,C 180,E1 19405.319,E2 19405.319} C_VEL
LIN {X 0,Y 497.642,Z 1015.596,A -85,B 0,C 180,E1 19404.36,E2 19404.36} C_VEL
LIN {X 0,Y 490.972,Z 1041.228,A -85,B 0,C 180,E1 19402.975,E2 19402.975} C_VEL
LIN {X 0,Y 484.511,Z 1063.253,A -85,B 0,C 180,E1 19401.557,E2 19401.557} C_VEL
LIN {X 0,Y 478.36,Z 1082.847,A -85,B 0,C 180,E1 19400.1,E2 19400.1} C_VEL
LIN {X 0,Y 472.288,Z 1101.146,A -85,B 0,C 180,E1 19398.548,E2 19398.548} C_VEL
LIN {X 0,Y 464.864,Z 1122.625,A -85,B 0,C 180,E1 19396.462,E2 19396.462} C_VEL
LIN {X 0,Y 457.202,Z 1143.536,A -85,B 0,C 180,E1 19394.068,E2 19394.068} C_VEL
LIN {X 0,Y 451.218,Z 1159.629,A -85,B 0,C 180,E1 19391.964,E2 19391.964} C_VEL
LIN {X 0,Y 445.624,Z 1174.591,A -85,B 0,C 180,E1 19389.758,E2 19389.758} C_VEL
LIN {X 0,Y 439.407,Z 1191.509,A -85,B 0,C 180,E1 19386.928,E2 19386.928} C_VEL
LIN {X 0,Y 433.501,Z 1207.628,A -85,B 0,C 180,E1 19383.776,E2 19383.776} C_VEL
LIN {X 0,Y 429.199,Z 1220.086,A -85,B 0,C 180,E1 19380.983,E2 19380.983} C_VEL
LIN {X 0,Y 425.634,Z 1231.101,A -85,B 0,C 180,E1 19378.181,E2 19378.181} C_VEL
LIN {X 0,Y 422.124,Z 1243.224,A -85,B 0,C 180,E1 19374.644,E2 19374.644} C_VEL
LIN {X 0,Y 419.546,Z 1253.287,A -85,B 0,C 180,E1 19371.098,E2 19371.098} C_VEL
LIN {X 0,Y 418.026,Z 1260.477,A -85,B 0,C 180,E1 19368.122,E2 19368.122} C_VEL
LIN {X 0,Y 417.04,Z 1266.256,A -85,B 0,C 180,E1 19365.297,E2 19365.297} C_VEL
LIN {X 0,Y 416.445,Z 1271.025,A -85,B 0,C 180,E1 19362.485,E2 19362.485} C_VEL
LIN {X 0,Y 416.094,Z 1274.643,A -85,B 0,C 180,E1 19359.829,E2 19359.829} C_VEL
LIN {X 0,Y 415.981,Z 1277.512,A -85,B 0,C 180,E1 19357.047,E2 19357.047} C_VEL
LIN {X 0,Y 415.932,Z 1279.433,A -85,B 0,C 180,E1 19354.28,E2 19354.28} C_VEL
LIN {X 0,Y 415.925,Z 1280.393,A -85,B 0,C 180,E1 19351.659,E2 19351.659} C_VEL
LIN {X 0,Y 415.901,Z 1280.488,A -85,B 0,C 180,E1 19348.904,E2 19348.904} C_VEL
LIN {X 0,Y 415.93,Z 1279.65,A -85,B 0,C 180,E1 19346.147,E2 19346.147} C_VEL
LIN {X 0,Y 415.97,Z 1277.875,A -85,B 0,C 180,E1 19343.381,E2 19343.381} C_VEL
LIN {X 0,Y 416.061,Z 1275.152,A -85,B 0,C 180,E1 19340.602,E2 19340.602} C_VEL
LIN {X 0,Y 416.407,Z 1271.413,A -85,B 0,C 180,E1 19337.77,E2 19337.77} C_VEL
LIN {X 0,Y 416.952,Z 1266.804,A -85,B 0,C 180,E1 19334.997,E2 19334.997} C_VEL
LIN {X 0,Y 417.911,Z 1261.128,A -85,B 0,C 180,E1 19332.174,E2 19332.174} C_VEL
LIN {X 0,Y 419.274,Z 1254.405,A -85,B 0,C 180,E1 19329.34,E2 19329.34} C_VEL
LIN {X 0,Y 421.182,Z 1246.594,A -85,B 0,C 180,E1 19326.503,E2 19326.503} C_VEL
LIN {X 0,Y 424.001,Z 1236.58,A -85,B 0,C 180,E1 19323.351,E2 19323.351} C_VEL
LIN {X 0,Y 428.438,Z 1222.442,A -85,B 0,C 180,E1 19319.582,E2 19319.582} C_VEL
LIN {X 0,Y 432.571,Z 1210.27,A -85,B 0,C 180,E1 19316.791,E2 19316.791} C_VEL
LIN {X 0,Y 437.173,Z 1197.338,A -85,B 0,C 180,E1 19314.17,E2 19314.17} C_VEL
LIN {X 0,Y 442.817,Z 1182.153,A -85,B 0,C 180,E1 19311.459,E2 19311.459} C_VEL
LIN {X 0,Y 450.063,Z 1162.76,A -85,B 0,C 180,E1 19308.478,E2 19308.478} C_VEL
LIN {X 0,Y 456.033,Z 1146.674,A -85,B 0,C 180,E1 19306.329,E2 19306.329} C_VEL
LIN {X 0,Y 461.922,Z 1130.594,A -85,B 0,C 180,E1 19304.423,E2 19304.423} C_VEL
LIN {X 0,Y 467.815,Z 1114.059,A -85,B 0,C 180,E1 19302.683,E2 19302.683} C_VEL
LIN {X 0,Y 474.388,Z 1094.95,A -85,B 0,C 180,E1 19300.909,E2 19300.909} C_VEL
LIN {X 0,Y 482.235,Z 1070.668,A -85,B 0,C 180,E1 19298.977,E2 19298.977} C_VEL
LIN {X 0,Y 488.285,Z 1050.357,A -85,B 0,C 180,E1 19297.595,E2 19297.595} C_VEL
LIN {X 0,Y 493.525,Z 1031.372,A -85,B 0,C 180,E1 19296.468,E2 19296.468} C_VEL
LIN {X 0,Y 498.616,Z 1011.352,A -85,B 0,C 180,E1 19295.441,E2 19295.441} C_VEL
LIN {X 0,Y 503.475,Z 990.145,A -85,B 0,C 180,E1 19294.509,E2 19294.509} C_VEL
LIN {X 0,Y 508.804,Z 963.59,A -85,B 0,C 180,E1 19293.545,E2 19293.545} C_VEL
LIN {X 0,Y 512.947,Z 937.924,A -85,B 0,C 180,E1 19292.82,E2 19292.82} C_VEL
LIN {X 0,Y 515.836,Z 915.968,A -85,B 0,C 180,E1 19292.335,E2 19292.335} C_VEL
LIN {X 0,Y 517.953,Z 893.291,A -85,B 0,C 180,E1 19291.925,E2 19291.925} C_VEL
LIN {X 0,Y 530.956,Z 675.486,A -85,B 0,C 180,E1 19288.543,E2 19288.543} C_VEL
LIN {X 0,Y 537.322,Z 571.291,A -85,B 0,C 180,E1 19286.903,E2 19286.903} C_VEL
LIN {X 0,Y 527.679,Z 555.399,A -85,B 0,C 180,E1 19284.28,E2 19284.28} C_VEL
LIN {X 0,Y 519.297,Z 542.271,A -85,B 0,C 180,E1 19281.697,E2 19281.697} C_VEL
LIN {X 0,Y 513.132,Z 533.126,A -85,B 0,C 180,E1 19279.553,E2 19279.553} C_VEL
LIN {X 0,Y 507.33,Z 524.576,A -85,B 0,C 180,E1 19277.255,E2 19277.255} C_VEL
LIN {X 0,Y 504.431,Z 520.835,A -85,B 0,C 180,E1 19275.994,E2 19275.994} C_VEL
LIN {X 0,Y 500.77,Z 515.971,A -85,B 0,C 180,E1 19274.217,E2 19274.217} C_VEL
LIN {X 0,Y 497.138,Z 511.312,A -85,B 0,C 180,E1 19272.192,E2 19272.192} C_VEL
LIN {X 0,Y 496.017,Z 510.175,A -85,B 0,C 180,E1 19271.512,E2 19271.512} C_VEL
LIN {X 0,Y 493.083,Z 506.698,A -85,B 0,C 180,E1 19269.454,E2 19269.454} C_VEL
LIN {X 0,Y 492.045,Z 504.662,A -85,B 0,C 180,E1 19268.531,E2 19268.531} C_VEL
LIN {X 0,Y 488.498,Z 501.384,A -85,B 0,C 180,E1 19264.696,E2 19264.696} C_VEL
LIN {X 0,Y 487.538,Z 498.466,A -85,B 0,C 180,E1 19262.351,E2 19262.351} C_VEL
LIN {X 0,Y 487.652,Z 498.59,A -85,B 0,C 180,E1 19256.826,E2 19256.826} C_VEL
LIN {X 0,Y 488.942,Z 502.036,A -85,B 0,C 180,E1 19254.131,E2 19254.131} C_VEL
LIN {X 0,Y 492.264,Z 505.018,A -85,B 0,C 180,E1 19250.766,E2 19250.766} C_VEL
LIN {X 0,Y 494.561,Z 508.772,A -85,B 0,C 180,E1 19248.926,E2 19248.926} C_VEL
LIN {X 0,Y 497.003,Z 511.022,A -85,B 0,C 180,E1 19247.392,E2 19247.392} C_VEL
LIN {X 0,Y 500.258,Z 515.512,A -85,B 0,C 180,E1 19245.532,E2 19245.532} C_VEL
LIN {X 0,Y 501.701,Z 517.142,A -85,B 0,C 180,E1 19244.806,E2 19244.806} C_VEL
LIN {X 0,Y 506.373,Z 523.15,A -85,B 0,C 180,E1 19242.652,E2 19242.652} C_VEL
LIN {X 0,Y 510.582,Z 528.675,A -85,B 0,C 180,E1 19240.94,E2 19240.94} C_VEL
LIN {X 0,Y 515.249,Z 534.879,A -85,B 0,C 180,E1 19239.228,E2 19239.228} C_VEL
LIN {X 0,Y 521.372,Z 543.139,A -85,B 0,C 180,E1 19237.207,E2 19237.207} C_VEL
LIN {X 0,Y 528.901,Z 553.812,A -85,B 0,C 180,E1 19234.976,E2 19234.976} C_VEL
LIN {X 0,Y 537.349,Z 566.278,A -85,B 0,C 180,E1 19232.729,E2 19232.729} C_VEL
LIN {X 0,Y 524.086,Z 782.129,A -85,B 0,C 180,E1 19229.383,E2 19229.383} C_VEL
LIN {X 0,Y 518.083,Z 880.695,A -85,B 0,C 180,E1 19227.842,E2 19227.842} C_VEL
LIN {X 0,Y 515.264,Z 908.067,A -85,B 0,C 180,E1 19227.306,E2 19227.306} C_VEL
LIN {X 0,Y 511.404,Z 934.261,A -85,B 0,C 180,E1 19226.606,E2 19226.606} C_VEL
LIN {X 0,Y 507.656,Z 955.445,A -85,B 0,C 180,E1 19225.903,E2 19225.903} C_VEL
LIN {X 0,Y 503.474,Z 975.891,A -85,B 0,C 180,E1 19225.092,E2 19225.092} C_VEL
LIN {X 0,Y 498.299,Z 998.181,A -85,B 0,C 180,E1 19224.05,E2 19224.05} C_VEL
LIN {X 0,Y 491.195,Z 1024.957,A -85,B 0,C 180,E1 19222.538,E2 19222.538} C_VEL
LIN {X 0,Y 485.429,Z 1044.536,A -85,B 0,C 180,E1 19221.231,E2 19221.231} C_VEL
LIN {X 0,Y 479.788,Z 1062.319,A -85,B 0,C 180,E1 19219.88,E2 19219.88} C_VEL
LIN {X 0,Y 473.733,Z 1080.268,A -85,B 0,C 180,E1 19218.334,E2 19218.334} C_VEL
